FUNCTION "mb_internal_s" : Bool   // FC23, SCL
{ S7_Optimized_Access := 'TRUE' }
VERSION : 0.1
   VAR_INPUT
      start : DInt;
      end : DInt;
   END_VAR
   VAR_IN_OUT
      buffer_lo : DInt;
      buffer_hi : DInt;
      q : "mb_query";
   END_VAR
   VAR_TEMP
      tmp : DInt;
   END_VAR
BEGIN
   // Internal function in the library for calculating
   // beginning and end for swapping.
   // 
   // This function dosen't work for discrete quries !

   // Find the beginning in the buffer where swaping should start.
   #buffer_lo := SEL(G := #start = 0,
                     IN0 := (#start - UDINT_TO_DINT(#q.z.q.data_addr)) * 2,
                     IN1 := 0);

   // Find end point in buffer.
   IF #end = 0 THEN  // Auto - Swap all words in query.
       #buffer_hi := #q.z.q.data_len * 2 - 1;

   ELSE // Address given for #end.
       #buffer_hi := (#end - UDINT_TO_DINT(#q.z.q.data_addr)) * 2 - 1 ;
   END_IF;

   // Test if there is valid input values.
   #mb_internal_s := #buffer_lo >= 0 AND #buffer_hi <= 249 ;

   // Error handling.
   IF NOT #mb_internal_s THEN // If not valid values.
       #q.stat.status := 16#fffe;
       #q.Error := #q.stat.error := true;
       #q.Done := #q.stat.done := false;
       #q.z.sb.log_data_addr := #q.z.q.data_addr;
   END_IF;
END_FUNCTION

// folder: Library/Modbus/Core/z/z internal testing functions/z Testing

FUNCTION_BLOCK "tcp_test"   // FB96, SCL
{ S7_Optimized_Access := 'TRUE' }
VERSION : 0.1
   VAR
      mb_query : "mb_query";
      mb_client_ctrl : "mb_client_ctrl";
      t1 : Word;
      t2 : Word;
      t3 : Word;
      t4 : Word;
      aa : Bool;
      mb_delay_between_queries : "mb_delay_between_queries";
      sb : "mb_station_block_udt";
   END_VAR
BEGIN

   #mb_client_ctrl.ip_addr[1] := 192;
   #mb_client_ctrl.ip_addr[2] := 168;
   #mb_client_ctrl.ip_addr[3] := 0;
   #mb_client_ctrl.ip_addr[4] := 33;
   #mb_client_ctrl(interface := 64,
                   conn_id := 123,
                   tcp_port := 502,
                   // timeout := T#500ms,
                   mb_query := #mb_query);

   #mb_delay_between_queries(// delay := T#1s,
                             mb_query := #mb_query);

   "mb_station_block_header"(sb := #sb, mb_query := #mb_query);

   #mb_query(mb_addr := 255,
             mode := #mb_query.c.write.holding_reg,
             data_addr := 1,
             data_ptr := #t1);

   #mb_query(mode := #mb_query.c.read.holding_reg,
             data_addr := 1,
             data_ptr := #t2);

   #mb_query(mode := #mb_query.c.write.holding_reg,
             data_addr := 2,
             data_ptr := #t2);

   #mb_query(mode := #mb_query.c.read.holding_reg,
             data_addr := 2,
             data_ptr := #t3);

   "mb_station_block_footer"(sb := #sb, mb_query := #mb_query);
END_FUNCTION_BLOCK

FUNCTION_BLOCK "rtu_test_1500"   // FB102, SCL
{ S7_Optimized_Access := 'TRUE' }
VERSION : 0.1
   VAR
      mb_master_1500_ctrl : "mb_master_1500_ctrl";
      mb_query : "mb_query";
      temperature_1 : "Jdrk_RS_WS_N01_8";
      temperature_2 : "Jdrk_RS_WS_N01_8";
      temperature_3 : "Jdrk_RS_WS_N01_8";
      sb_temp_no_answer_1 : "sb_temp_no_answer";
      sb_temp_no_answer_2 : "sb_temp_no_answer";
      sb_temp_no_answer_3 : "sb_temp_no_answer";
      sb_temp_error_1 : "sb_temp_error";
      sb_temp_error_2 : "sb_temp_error";
      sb_temp_error_3 : "sb_temp_error";
      delay_between_queries : "mb_delay_between_queries";
      mb_delay : "mb_delay";
   END_VAR
BEGIN

   #mb_master_1500_ctrl.conf.parity := 0;
   #mb_master_1500_ctrl(hardware_id := 269,
                        operating_mode := 4,
                        baud := 9600,
                        mb_query := #mb_query);

   #delay_between_queries(mb_query := #mb_query);


   #temperature_1(mb_query := #mb_query);
   #temperature_2(mb_query := #mb_query);
   #temperature_3(mb_query := #mb_query);

   #mb_delay(mb_query := #mb_query);

   #sb_temp_no_answer_1(mb_query := #mb_query);
   #sb_temp_no_answer_2(mb_query := #mb_query);
   #sb_temp_no_answer_3(mb_query := #mb_query);

   #sb_temp_error_1(mb_query := #mb_query);
   #sb_temp_error_2(mb_query := #mb_query);
   #sb_temp_error_3(mb_query := #mb_query);
END_FUNCTION_BLOCK

FUNCTION_BLOCK "rtu_test2_1200"   // FB115, SCL
{ S7_Optimized_Access := 'TRUE' }
VERSION : 0.1
   VAR
      mb_query : "mb_query";
      mb_master_1200_ctrl : "mb_master_1200_ctrl";
      Danfoss : "Danfoss_VLT";
      Mjk_expert_1 : "Mjk_expert";
      Mjk_expert_2 : "Mjk_expert";
      Mjk_expert_3 : "Mjk_expert";
   END_VAR
BEGIN
   #mb_master_1200_ctrl.conf.parity := 0;
   #mb_master_1200_ctrl(hardware_id := 0, // "Local~CB_1241_(RS485)",
                        baud := 9600,
                        mb_query := #mb_query);

   #Mjk_expert_1(mb_addr := 1, mb_query := #mb_query);
   #Mjk_expert_2(mb_addr := 1, mb_query := #mb_query);
   #Mjk_expert_3(mb_addr := 1, mb_query := #mb_query);

   #Danfoss(mb_addr := 2, mb_query := #mb_query);
END_FUNCTION_BLOCK

FUNCTION_BLOCK "rtu_test1_1200"   // FB116, SCL
{ S7_Optimized_Access := 'TRUE' }
VERSION : 0.1
   VAR
      mb_query : "mb_query";
      mb_master_1200_ctrl : "mb_master_1200_ctrl";
      delay_between_queries : "mb_delay_between_queries";
      delay : "mb_delay";
      __ : Bool;
      temperature_1 : "Jdrk_RS_WS_N01_8";
      temperature_2 : "Jdrk_RS_WS_N01_8";
      temperature_3 : "Jdrk_RS_WS_N01_8";
      sb_temp_no_answer_1 : "sb_temp_no_answer";
      sb_temp_no_answer_2 : "sb_temp_no_answer";
      sb_temp_no_answer_3 : "sb_temp_no_answer";
      sb_temp_error_1 : "sb_temp_error";
      sb_temp_error_2 : "sb_temp_error";
      sb_temp_error_3 : "sb_temp_error";
      _ : Bool;
      bool_arrary : Array[0..15] of Bool;
      sb : "mb_station_block_udt";
   END_VAR
BEGIN
   #mb_master_1200_ctrl.conf.parity := 0;
   #mb_master_1200_ctrl(hardware_id := 269, // "Local~CB_1241_(RS485)",
                        baud := 9600,
                        mb_query := #mb_query);

   #delay_between_queries(mb_query := #mb_query);

   #temperature_1(mb_query := #mb_query);
   #temperature_2(mb_query := #mb_query);
   #temperature_3(mb_query := #mb_query);

   #delay(mb_query := #mb_query);

   #sb_temp_no_answer_1(mb_query := #mb_query);
   #sb_temp_no_answer_2(mb_query := #mb_query);
   #sb_temp_no_answer_3(mb_query := #mb_query);

   #sb_temp_error_1(mb_query := #mb_query);
   #sb_temp_error_2(mb_query := #mb_query);
   #sb_temp_error_3(mb_query := #mb_query);

   "mb_station_block_header"(sb := #sb, mb_query := #mb_query);
   #mb_query.mb_addr := 1;
   #mb_query.mode := #mb_query.c.read.input_reg;
   #mb_query.data_addr := 1;
   "mb_query_bits"(data_ptr := #bool_arrary, mb_query := #mb_query);
   "mb_station_block_footer"(sb := #sb, mb_query := #mb_query);
END_FUNCTION_BLOCK

// folder: Library/Modbus/Core/z/z internal testing functions/z Testing/nolib

FUNCTION_BLOCK "client"   // FB112, SCL
{ S7_Optimized_Access := 'TRUE' }
VERSION : 0.1
   VAR
      client : MB_CLIENT;
      tcon_ip_v4 : TCON_IP_v4;
      buffer : Array[0..3] of Byte;
      rtrig_err : R_TRIG;
      rtrig_busy : R_TRIG;
      rtrig_done : R_TRIG;
      err_cnt : UDInt;
      busy_cnt : UDInt;
      done_cnt : UDInt;
      a4 : USInt;
   END_VAR
BEGIN
   #tcon_ip_v4.InterfaceId := 64;
   #tcon_ip_v4.ID := 456;
   #tcon_ip_v4.ConnectionType := 11; // tcp
   #tcon_ip_v4.ActiveEstablished := true;
   #tcon_ip_v4.RemoteAddress.ADDR[1] := 192;
   #tcon_ip_v4.RemoteAddress.ADDR[2] := 168;
   #tcon_ip_v4.RemoteAddress.ADDR[3] := 0;
   #tcon_ip_v4.RemoteAddress.ADDR[4] := #a4;
   #tcon_ip_v4.RemotePort := 502;

   #client(REQ := #client.REQ,
           DISCONNECT := #client.DISCONNECT,
           MB_MODE := 103,
           MB_DATA_ADDR := 1000,
           MB_DATA_LEN := 1,
           MB_DATA_PTR := #buffer,
           CONNECT := #tcon_ip_v4);

   #rtrig_err(CLK := #client.ERROR);
   #err_cnt += BOOL_TO_UINT( #rtrig_err.Q );

   #rtrig_busy(CLK := #client.BUSY);
   #busy_cnt += BOOL_TO_UINT(#rtrig_busy.Q);

   #rtrig_done(CLK := #client.DONE);
   #done_cnt += BOOL_TO_UINT(#rtrig_done.Q);
END_FUNCTION_BLOCK

// folder: Library/Modbus/Core/z/z internal testing functions/z Testing/sb

FUNCTION_BLOCK "sb_temp_no_answer"   // FB32, SCL
{ S7_Optimized_Access := 'TRUE' }
VERSION : 0.1
   VAR_OUTPUT
      Temperature : Real;
   END_VAR
   VAR_IN_OUT
      mb_query : "mb_query";
   END_VAR
   VAR
      sb : "mb_station_block_udt";
   END_VAR
   VAR RETAIN
      offset : Real;
   END_VAR
   VAR_TEMP
      tmp : Int;
   END_VAR
BEGIN
   // JDRK - RS-WS-N01-8 - Temperature and Humidity sensor

   "mb_station_block_header"(sb := #sb, mb_query := #mb_query);

   #mb_query(mb_addr := 200,
             mode := #mb_query.c.read.input_reg,
             data_addr := 1,
             data_ptr := #tmp);

   IF #mb_query.Done THEN
       #Temperature := INT_TO_REAL(#tmp) / 10 + #offset;
   END_IF;

   "mb_station_block_footer"(sb := #sb, mb_query := #mb_query);
END_FUNCTION_BLOCK

FUNCTION_BLOCK "sb_temp_error"   // FB33, SCL
{ S7_Optimized_Access := 'TRUE' }
VERSION : 0.1
   VAR_OUTPUT
      Temperature : Real;
   END_VAR
   VAR_IN_OUT
      mb_query : "mb_query";
   END_VAR
   VAR
      sb : "mb_station_block_udt";
   END_VAR
   VAR RETAIN
      tt : Array[0..100] of Int;
   END_VAR
   VAR_TEMP
      tmp : Int;
   END_VAR
BEGIN
   // JDRK - RS-WS-N01-8 - Temperature and Humidity sensor

   "mb_station_block_header"(sb := #sb, mb_query := #mb_query);

   #mb_query(mb_addr := 1,
             mode := #mb_query.c.read.input_reg,
             data_addr := 1,
             data_ptr := #tmp);

   IF #mb_query.Done THEN
       #Temperature := INT_TO_REAL(#tmp) / 10;
   END_IF;

   // Query producing a error.
   #mb_query(mb_addr := 1,
             mode := #mb_query.c.read.input_reg,
             data_addr := 1,
             data_ptr := #tt);

   "mb_station_block_footer"(sb := #sb, mb_query := #mb_query);
END_FUNCTION_BLOCK

// folder: Library/Modbus/Core/z Special code snippets examples/Not needed for regular users

FUNCTION_BLOCK "Example Done and error"   // FB56, SCL
{ S7_Optimized_Access := 'TRUE' }
VERSION : 0.1
   VAR_IN_OUT
      mb_query : "mb_query";
   END_VAR
   VAR
      query1_data : Word;
      done_cnt : UInt;
      query2_data : Word;
   END_VAR
BEGIN
   // To get information about when a particular query has executed.

   #mb_query(mb_addr := 123,
             mode := #mb_query.c.write.holding_reg,
             data_addr := 456,
             data_ptr := #query1_data);

   // The if-statement bellow has to be put after the particular 
   // query, and before the next query.    

   IF #mb_query.Done THEN
       // Some action after a successfully query.    
       #done_cnt += 1; // Eg. count successfully queries.

   ELSIF #mb_query.Error THEN
       // Some action if a faild query.    

       // #mb_query.stat.status , gives more information about 
       // the error.         

       IF #mb_query.stat.error_comm THEN
           ; // Some particular action if communication error.
       END_IF;

   END_IF;

   // Next query...
   #mb_query(mb_addr := 111,
             mode := #mb_query.c.read.holding_reg,
             data_addr := 789,
             data_ptr := #query2_data);
END_FUNCTION_BLOCK

FUNCTION_BLOCK "Example Swap"   // FB78, SCL
{ S7_Optimized_Access := 'TRUE' }
VERSION : 0.1
   VAR_IN_OUT
      mb_query : "mb_query";
   END_VAR
   VAR
      static_tmp_var : DWord;
      value : DWord;
      value2 : DWord;
      value_real_1 : Real;
      value_real_2 : Real;
   END_VAR
   VAR_TEMP
      "e" : Int;
      param : "mb_set_udt";
   END_VAR
   VAR CONSTANT
      ALL : Int;
   END_VAR
BEGIN
   // For some modbus devices, when two registers are combined into one,
   // the data is stored as little endian, not big endian like Siemens 
   // PLC does. To solve this, the SWAP function needs to be utilized.
   #mb_query(mb_addr := 123,
             mode := #mb_query.c.read.holding_reg,
             data_addr := 123,
             data_ptr := #static_tmp_var);

   #value := SWAP(#static_tmp_var);


   // For other device, when two registers are combined, the least significant 
   // word is stored first and the most significant word is stored in the 
   // following register. When this is the case, the ROR-function needs 
   // to be used.
   #mb_query(mb_addr := 123,
             mode := #mb_query.c.read.holding_reg,
             data_addr := 123,
             data_ptr := #static_tmp_var);

   #value := ROR(IN := #static_tmp_var, N := 16);


   // In some situation both SWAP and ROR need to be used.
   #mb_query(mb_addr := 123,
             mode := #mb_query.c.read.holding_reg,
             data_addr := 123,
             data_ptr := #static_tmp_var);

   #value := SWAP(ROR(IN := #static_tmp_var, N := 16));

   // How the data is stored, is usually described in the
   // data sheet of each device.

   // ========================================================================

   // The code bellow it's anather approach. It may be har understand, but it 
   // should be okay to understand what it do.

   IF "mb_query_range"(start := 100, end := 150, q := #mb_query) THEN
       #"e" := "mb_swap_word"(start := #ALL, end := #ALL, q := #mb_query);
       #"e" := "mb_read_buffer"(addr := 100, ptr := #value, q := #mb_query);
       #"e" := "mb_read_buffer"(addr := 120, ptr := #value2, q := #mb_query);
   END_IF;

   IF "mb_query_range"(start := 200, end := 250, q := #mb_query) THEN
       #param.double := true; // 4 bytes
       #param.factor := 10; // 
       #value_real_1 := "mb_buffer_get"(addr := 200, param := #param, q := #mb_query);
       #value_real_2 := "mb_buffer_get"(addr := 220, param := #param, q := #mb_query);
   END_IF;
END_FUNCTION_BLOCK

FUNCTION_BLOCK "Example Read first"   // FB85, SCL
{ S7_Optimized_Access := 'TRUE' }
VERSION : 0.1
   VAR_INPUT
      input1 : Bool;
      input2 : Bool;
   END_VAR
   VAR_IN_OUT
      mb_query : "mb_query";
   END_VAR
   VAR
      write : Bool;
      data : Word;
   END_VAR
BEGIN
   // Sometimes only some bits in a word need to be manipulated, 
   // without touching the other bits, bellow is an example how 
   // that can be achieved.

   #mb_query.mb_addr := 123;
   #mb_query.data_addr := 456;

   IF #write THEN // (Initially false)

       // Manipulating only bit 5 and 11
       #data.%X5 := #input1;
       #data.%X11 := #input2;

       #mb_query(mode := #mb_query.c.write.holding_reg,
                 data_ptr := #data);

   ELSE // read the register before write to the same one.
       #mb_query(mode := #mb_query.c.read.holding_reg,
                 data_ptr := #data);

       // Has query above been executed successfully?
       IF #mb_query.Done THEN
           #write := true;
       END_IF;

   END_IF;

   // Note: The read only option (#sb.conf.read_conly) can't be
   // used when the metod above is used.
END_FUNCTION_BLOCK

FUNCTION_BLOCK "Example Forced execution order"   // FB89, SCL
{ S7_Optimized_Access := 'TRUE' }
VERSION : 0.1
   VAR_IN_OUT
      mb_query : "mb_query";
   END_VAR
   VAR
      state : Int;
      query_1 : Word;
      query_2 : UInt;
      query_3 : Word;
      query_4 : Word;
   END_VAR
BEGIN
   // If the execution need to be forced to a given order, then the 
   // example bellow can be followed.

   CASE #state OF

       0:  // 1st query
           #mb_query(mb_addr := 123,
                     mode := #mb_query.c.write.holding_reg,
                     data_addr := 123,
                     data_ptr := #query_1);
           #state += BOOL_TO_SINT(#mb_query.Done);
           // «#mb_query.done» is set true when the query above is done 
           // successfully. When next query is executed, «#mb_query.done»
           // is set back false.

       1:  // 2nd query
           #mb_query(mb_addr := 123,
                     mode := #mb_query.c.write.holding_reg,
                     data_addr := 456,
                     data_ptr := #query_2);
           #state += BOOL_TO_SINT(#mb_query.Done);

       2:  // 3rd query
           #mb_query(mb_addr := 123,
                     mode := #mb_query.c.read.holding_reg,
                     data_addr := 789,
                     data_ptr := #query_3);
           IF #mb_query.Done THEN
               #state := 0;
           END_IF;

   END_CASE;

   // 4th query, this query is executed three times as often 
   // as the queries above.
   #mb_query(mb_addr := 123,
             mode := #mb_query.c.read.input_reg,
             data_addr := 1234,
             data_ptr := #query_4);


   // If the state machine has both read and write queries then
   // #sb.conf.read_only can't be used.
END_FUNCTION_BLOCK

FUNCTION_BLOCK "Example discrete queries"   // FB101, SCL
{ S7_Optimized_Access := 'TRUE' }
VERSION : 0.1
   VAR_IN_OUT
      mb_query : "mb_query";
   END_VAR
   VAR
      one_bool : Bool;
      two_bools : Struct
         b1 : Bool;
         b2 : Bool;
      END_STRUCT;
   END_VAR
BEGIN
   // Discrete queries.

   // When doing discrete queries the data_len parameter need to
   // be specified manualy.
   #mb_query(mb_addr := 123,
             mode := #mb_query.c.read.discrete_input,
             data_addr := 456,
             data_len := 1,
             data_ptr := #one_bool); // A single boolean.

   // Another quering two bool's
   #mb_query(mb_addr := 123,
             mode := #mb_query.c.read.discrete_input,
             data_addr := 789,
             data_len := 2,
             data_ptr := #two_bools); // A struct with two boolean inside.

   // After discrete queries, data_len should be set back in to auto.
   #mb_query.data_len := #mb_query.c.auto_len;
END_FUNCTION_BLOCK

FUNCTION_BLOCK "Example sequence"   // FB103, SCL
{ S7_Optimized_Access := 'TRUE' }
VERSION : 0.1
   VAR_INPUT
      mb_addr : USInt;
   END_VAR
   VAR_IN_OUT
      mb_query : "mb_query";
   END_VAR
   VAR
      sb : "mb_station_block_udt";
      sequence : "mb_sequence";
      read1 : Word;
      read2 : Word;
      read3 : Word;
      write1 : Word;
      write2 : Word;
      write3 : Word;
   END_VAR
BEGIN
   "mb_station_block_header"(sb := #sb, mb_query := #mb_query);
   #mb_query.mb_addr := #mb_addr;

   // High priority queries:
   #mb_query(mode := #mb_query.c.read.holding_reg,
             data_addr := 12345,
             data_ptr := #write3);

   IF #sequence.Done THEN
       #mb_query(mode := #mb_query.c.write.holding_reg,
                 data_addr := 54321,
                 data_ptr := #write3);
   END_IF;

   // Low priority queries:
   // Some queries that doesn't need to be run so often, the state
   // machines bellow make low priority queries be executed less often.
   #sequence.conf.first_state := 1600;
   CASE "mb_sequence_init"(sequence := #sequence, mb_query := #mb_query) OF
           // --------- Read holding reg queries (3xx) ---------
       300: #mb_query(data_addr := 123, data_ptr := #read1);
       301: #mb_query(data_addr := 456, data_ptr := #read2);
       302: #mb_query(data_addr := 789, data_ptr := #read3);

           #sequence.next_state := 1600;
           // --------- Write holding reg queries (16xx) ---------     
       1600: #mb_query(data_addr := 654, data_ptr := #write1);
       1601: #mb_query(data_addr := 321, data_ptr := #write2);
           #sequence.next_state := 300;
       ELSE
           #sequence.state += 1;
   END_CASE;
   #sequence(sb := #sb, mb_query := #mb_query);

   "mb_station_block_footer"(sb := #sb, mb_query := #mb_query);
END_FUNCTION_BLOCK

// folder: Library/Modbus/Docs

FUNCTION "mb_version" : String   // FC6, SCL
{ S7_Optimized_Access := 'TRUE' }
VERSION : 0.1
BEGIN
   // Library version.
   #mb_version := '3.2.0';

   (*

   www.rexhip.com


   Copyright (c) 2018 Ola Bjørnli 

   Permission is hereby granted, free of charge, to any person obtaining a copy
   of this software and associated documentation files (the "Software"), to deal
   in the Software without restriction, including without limitation the rights
   to use, copy, modify, merge, publish, distribute, sublicense, and/or sell
   copies of the Software, and to permit persons to whom the Software is
   furnished to do so, subject to the following conditions:

   The above copyright notice and this permission notice shall be included in all
   copies or substantial portions of the Software.

   THE SOFTWARE IS PROVIDED "AS IS", WITHOUT WARRANTY OF ANY KIND, EXPRESS OR
   IMPLIED, INCLUDING BUT NOT LIMITED TO THE WARRANTIES OF MERCHANTABILITY,
   FITNESS FOR A PARTICULAR PURPOSE AND NONINFRINGEMENT. IN NO EVENT SHALL THE
   AUTHORS OR COPYRIGHT HOLDERS BE LIABLE FOR ANY CLAIM, DAMAGES OR OTHER
   LIABILITY, WHETHER IN AN ACTION OF CONTRACT, TORT OR OTHERWISE, ARISING FROM,
   OUT OF OR IN CONNECTION WITH THE SOFTWARE OR THE USE OR OTHER DEALINGS IN THE
   SOFTWARE.

   *)
END_FUNCTION

FUNCTION "mb_Debugging" : Void   // FC15, SCL
{ S7_Optimized_Access := 'TRUE' }
VERSION : 0.1
BEGIN
   (* 
   # General debugging:
   - Look online and check that the latest version of the library 
     is in use. (www.rexhip.com or github.com/rexhip/rexhip)
   - All queries need to be executed in same order, this implicates 
     that it's NOT possible to put some queries in interupts and 
     other in cyclic OB's, this would interfere with the order.
   - Look inside the data blcok of the SB of the device that having 
     problem, and locate «#sb.log...», see if the counters are 
     running and lookup the error code of «#sb.log.error_status», 
     «#sb.log.error_data_addr» will tell witch query generating the 
     error. 
   - Try reboot PLC.

   # Modbus RTU
   - Try to increase timeout, repeaters on the bus need additional 
     time.
   - All the devies on the bus need to have a unique address.
   - Parity, buard rate, stop bits need to be the same in all 
     devices. The modbus specification state on page 20, that 19200
     is the default/recommended buad rate. The specification also 
     state, on page 12, that parity should be "even".
   - Electrical polarity, for some devices the connection "A" and "B" 
     is mislabeled, try to swap them.
   - Check for correct hardware id,

   # Modbus TCP
   - Try to increase timeout, creating a TCP-connection may take long.
   - Check IP-address.
   - Check TCP-port, 502 is default.
   - Check for unic connection-id.
   - Try set unit address to 255, (not for gateways)

   # Station Blocks 
   - If mb_station_block_header has executed in one block then 
     mb_station_block_foother also need to be executed. Cheack that 
     there is no RETURN or simular between them.
   - Check datasheet of device for special requirement: function codes 
     supported, max data length, register required to be queried 
     together, etc.  
   - A query can't be longer then 124 words.   
   - Try to comment out queries and see if it solve the problem.  

   # TIA-portal upgrading firmware error
     If you upgrade the firmware of a plc in a project, several errors in 
     the code regarding in serialize and deserialize will appear. This is 
     due to a error in TIA-portal. The solution is avoid using the upgrade 
     function, and rather add a new plc in the project and move all 
     elements to the new plc.

   # Some status codes and solutions:
     8188:     Try upgrade to latest version of the library. 

   # Customs status error codes
   - ffff: mb_read_buffer:     The request data is not avalible inside the 
                               buffer. check value of #addr.                            
   - fffe:                     
   - fffd: mb_buffer_get       The request data is not avalible inside the 
                               buffer. check value of #addr.

   *)
END_FUNCTION

// folder: Library/Modbus/Station blocks/sb Tested/Danfoss

FUNCTION_BLOCK "Danfoss_VLT"   // FB71, SCL
{ S7_Optimized_Access := 'TRUE' }
VERSION : 0.1
   VAR_INPUT
      mb_addr : USInt;
   END_VAR
   VAR_IN_OUT
      mb_query : "mb_query";
   END_VAR
   VAR
      sb : "mb_station_block_udt";
   END_VAR
   VAR RETAIN
      conf : Struct
         Send_config_to_drive : Bool := true;
         auto_start : Bool;
         action_no_communication : Int := 2;   // 2: Stop,
         input_source : Int := 2;   // 2: ctw fieldbus
      END_STRUCT;
   END_VAR
   VAR
      data : "variable_frequency_drive_udt";
      alarm_word : DWord;
      read : Struct   // (unscaled)
         stw : Struct   // Status word
            speed_eq_reference : Bool;   // [08]
            bus_control : Bool;   // [09] false=hand mode
            frequency_limit_ok : Bool;   // [10]
            in_operation : Bool;   // [11]
            stopped_auto_start : Bool;   // [12]
            voltage_exceeded : Bool;   // [13]
            torque_exceeded : Bool;   // [14]
            timer_exceeded : Bool;   // [15]
            control_ready : Bool;   // [00]
            drive_ready : Bool;   // [01]
            enable : Bool;   // [02] 0=Coasting
            trip : Bool;   // [03]
            error_no_trip : Bool;   // [04]
            x05 : Bool;   // [05]
            triplock : Bool;   // [06]
            warning : Bool;   // [07]
         END_STRUCT;
         man : Int;   // man actual value
      END_STRUCT;
      write : Struct   // Controll word
         ctw : Struct   // Controll word
            x08 : Bool;   // [08]
            use_ramp_2 : Bool;   // [09]
            data_valid : Bool := TRUE;   // [10]
            x11 : Bool;   // [11]
            x12 : Bool;   // [12]
            x13 : Bool;   // [13]
            x14 : Bool;   // [14]
            reverse : Bool;   // [15]
            x00 : Bool;   // [00]
            x01 : Bool;   // [01]
            dc_break_NOT : Bool := TRUE;   // [02]
            coast_NOT : Bool := TRUE;   // [03]
            quick_stop_NOT : Bool := TRUE;   // [04]
            hold_output_frequency_NOT : Bool := TRUE;   // [05]
            start : Bool;   // [06]
            reset : Bool;   // [07]
         END_STRUCT;
         ref : Int;
      END_STRUCT;
      sequence : "mb_sequence";
   END_VAR
   VAR_TEMP
      tmp : Int;
      dtmp : DInt;
   END_VAR
BEGIN
   (*  Danfoss - VLT
       doc_MG20N202.pdf, doc_MG20O602.pdf

       8.4 : Action if no communication.    (2=stop)     
       8.1 : Select input source            (2=CTW=fieldbus)     
   *)
   "mb_station_block_header"(sb := #sb, mb_query := #mb_query);
   #mb_query.mb_addr := #mb_addr;

   REGION Low priority queries
       // Some queries that doesn't need to be run so often, the state machines
       // bellow make low priority queries be executed less often.
       #sequence.conf.first_state := SEL(G := #conf.Send_config_to_drive,
                                         IN0 := 300, IN1 := 1600);
       CASE "mb_sequence_init"(sequence := #sequence, mb_query := #mb_query) OF
               // --------- Read holding reg queries ---------
           300:  // Frequency (hz)
               #mb_query(data_addr := "p"(a := 16, b := 13), data_ptr := #tmp);
               IF #mb_query.Done THEN
                   #data.out.frequency := DINT_TO_REAL(#tmp) * 0.1;
               END_IF;
           301:  // Electrical current 
               #mb_query(data_addr := "p"(a := 16, b := 14), data_ptr := #dtmp);
               IF #mb_query.Done THEN
                   #data.out.current := DINT_TO_REAL(#dtmp) * 0.01;
               END_IF;
           302:  // RPM
               #mb_query(data_addr := "p"(a := 16, b := 17), data_ptr := #dtmp);
               IF #mb_query.Done THEN
                   #data.out.rpm := DINT_TO_REAL(#dtmp) / 60;
               END_IF;
           303:  // Power
               #mb_query(data_addr := "p"(a := 16, b := 10), data_ptr := #dtmp);
               IF #mb_query.Done THEN
                   #data.out.power := DINT_TO_REAL(#dtmp) * 10;
               END_IF;
           304:  // Heatsink Temp. 
               #mb_query(data_addr := "p"(a := 16, b := 34), data_ptr := #tmp);
               IF #mb_query.Done THEN
                   #data.out.heatsing_temperature := #tmp;
               END_IF;
           305:  // Motor voltage
               #mb_query(data_addr := "p"(a := 16, b := 12), data_ptr := #tmp);
               IF #mb_query.Done THEN
                   #data.out.voltage := INT_TO_REAL(#tmp) * 0.1;
               END_IF;
           306:  // Alarm word 
               #mb_query(data_addr := "p"(a := 16, b := 92), data_ptr := #dtmp);
               IF #mb_query.Done THEN
                   #alarm_word := DINT_TO_DWORD(#dtmp);
               END_IF;
           307:  // Torque [%] 
               #mb_query(data_addr := "p"(a := 16, b := 22), data_ptr := #tmp);
               IF #mb_query.Done THEN
                   #data.out.torque_percent := #tmp;
               END_IF;
               #sequence.next_state := #sequence.conf.first_state;

               // --------- Write holding reg queries ---------     
           1600: // Action if no communication. (2=stop)     
               #mb_query(data_addr := "p"(a := 8, b := 4),
                         data_ptr := #conf.action_no_communication);
           1601: // Select input source (2=CTW=fieldbus)     
               #mb_query(data_addr := "p"(a := 8, b := 1),
                         data_ptr := #conf.input_source);
               #sequence.next_state := 300;
           ELSE
               #sequence.state += 1;
       END_CASE;
       #sequence(sb := #sb, mb_query := #mb_query);
   END_REGION

   REGION High priority queries
       // Status word  and main actual value 
       #mb_query(mode := #mb_query.c.read.holding_reg,
                 data_addr := 2909,
                 data_ptr := #read);
       IF #mb_query.Done THEN
           #data.out.ready := #read.stw.control_ready
           (* *)AND #read.stw.drive_ready AND #read.stw.bus_control;
           #data.out.error := #read.stw.trip OR #read.stw.error_no_trip;
           #data.out.auto := #read.stw.bus_control;
           #data.out.in_operation := #read.stw.in_operation;
           #data.out.output_percent := INT_TO_REAL(#read.man) / 16#4000 * 100;
       END_IF;
       // Send ctw and ref
       #write.ctw.reset := #data.in.reset;
       #write.ctw.dc_break_NOT := NOT #data.in.dc_break;
       #write.ctw.coast_NOT := NOT #data.in.cost;
       #write.ctw.quick_stop_NOT := NOT #data.in.quick_stop;
       #write.ctw.start := #data.in.start;
       #write.ref := REAL_TO_INT(#data.in.ref / 100 * 16#4000);
       #mb_query(mode := #mb_query.c.write.holding_reg,
                 data_addr := 2809,
                 data_ptr := #write);
   END_REGION

   "mb_station_block_footer"(sb := #sb, mb_query := #mb_query);

   (* Terminals:
   68  RS485 D+
   69  RS485 D-
   *)
END_FUNCTION_BLOCK

FUNCTION_BLOCK "Danfoss_VLT_simple"   // FB124, SCL
{ S7_Optimized_Access := 'TRUE' }
VERSION : 0.1
   VAR_INPUT
      mb_addr : USInt;
      ref : Real;
      start : Bool;
      cost : Bool;
      dc_break : Bool;
      quick_stop : Bool;
   END_VAR
   VAR_OUTPUT
      Ready : Bool;
      Feedback : Real;
   END_VAR
   VAR_IN_OUT
      mb_query : "mb_query";
   END_VAR
   VAR
      sb : "mb_station_block_udt";
      data : "variable_frequency_drive_udt";
      read : Struct   // (unscaled)
         stw : Struct   // Status word
            speed_eq_reference : Bool;   // [08]
            bus_control : Bool;   // [09] false=hand mode
            frequency_limit_ok : Bool;   // [10]
            in_operation : Bool;   // [11]
            stopped_auto_start : Bool;   // [12]
            voltage_exceeded : Bool;   // [13]
            torque_exceeded : Bool;   // [14]
            timer_exceeded : Bool;   // [15]
            control_ready : Bool;   // [00]
            drive_ready : Bool;   // [01]
            enable : Bool;   // [02] 0=Coasting
            trip : Bool;   // [03]
            error_no_trip : Bool;   // [04]
            x05 : Bool;   // [05]
            triplock : Bool;   // [06]
            warning : Bool;   // [07]
         END_STRUCT;
         man : Int;   // man actual value
      END_STRUCT;
      write : Struct   // Controll word
         ctw : Struct   // Controll word
            x08 : Bool;   // [08]
            use_ramp_2 : Bool;   // [09]
            data_valid : Bool := TRUE;   // [10]
            x11 : Bool;   // [11]
            x12 : Bool;   // [12]
            x13 : Bool;   // [13]
            x14 : Bool;   // [14]
            reverse : Bool;   // [15]
            x00 : Bool;   // [00]
            x01 : Bool;   // [01]
            dc_break_NOT : Bool := TRUE;   // [02]
            coast_NOT : Bool := TRUE;   // [03]
            quick_stop_NOT : Bool := TRUE;   // [04]
            hold_output_frequency_NOT : Bool := TRUE;   // [05]
            start : Bool;   // [06]
            reset : Bool;   // [07]
         END_STRUCT;
         ref : Int;
      END_STRUCT;
   END_VAR
BEGIN
   (*  Danfoss - VLT
       doc_MG20N202.pdf, doc_MG20O602.pdf

       8.4 : Action if no communication.    (2=stop)     
       8.1 : Select input source            (2=CTW=fieldbus)     

       Terminals:
       68  RS485 D+
       69  RS485 D-
   *)
   "mb_station_block_header"(sb := #sb, mb_query := #mb_query);
   #mb_query.mb_addr := #mb_addr;

   // Status word  and main actual value 
   #mb_query(mode := #mb_query.c.read.holding_reg,
             data_addr := 2909,
             data_ptr := #read);
   IF #mb_query.Done THEN
       #Ready := #read.stw.control_ready
       (* *)AND #read.stw.drive_ready AND #read.stw.bus_control;
       #Feedback := INT_TO_REAL(#read.man) / 16#4000 * 100;
   END_IF;

   // Send ctw and ref
   #write.ctw.dc_break_NOT := NOT #dc_break;
   #write.ctw.coast_NOT := NOT #cost;
   #write.ctw.quick_stop_NOT := NOT #quick_stop;
   #write.ctw.start := #start;
   #write.ref := REAL_TO_INT(#ref / 100 * 16#4000);
   #mb_query(mode := #mb_query.c.write.holding_reg,
             data_addr := 2809,
             data_ptr := #write);

   "mb_station_block_footer"(sb := #sb, mb_query := #mb_query);
END_FUNCTION_BLOCK

FUNCTION "p" : UInt   // FC14, SCL
{ S7_Optimized_Access := 'TRUE' }
VERSION : 0.1
   VAR_INPUT
      "a" : USInt;
      "b" : USInt;
   END_VAR
BEGIN
   // Calculation data_addr for danfoss vlt.

   #p := USINT_TO_UINT(#"a") * 1000
   (* *)+ USINT_TO_UINT(#"b") * 10
   (* *)- 1;
END_FUNCTION

// folder: Library/Modbus/Station blocks/sb Tested/MJK

FUNCTION_BLOCK "Mjk_expert"   // FB35, SCL
{ S7_Optimized_Access := 'TRUE' }
VERSION : 0.1
   VAR_INPUT
      mb_addr : USInt;
   END_VAR
   VAR_IN_OUT
      mb_query : "mb_query";
   END_VAR
   VAR
      sb : "mb_station_block_udt";
      data : Struct
         pressure : Real;
         temperature : Real;
      END_STRUCT;
   END_VAR
BEGIN
   // MJK - Expert 700-7060-7070 - Pressure transmitters

   "mb_station_block_header"(sb := #sb, mb_query := #mb_query);
   #mb_query.mb_addr := #mb_addr;

   #mb_query.mode := #mb_query.c.read.holding_reg;
   #mb_query(data_addr := 16#100, data_ptr := #data);

   "mb_station_block_footer"(sb := #sb, mb_query := #mb_query);

   (*
       Rød     +24V
       Brown   GND
       Yellow  RS485 B
       Gray    RS485 A
       White   Voltage output
   *)
END_FUNCTION_BLOCK

// folder: Library/Modbus/Station blocks/sb Tested/Ponsel mesure

FUNCTION_BLOCK "Ponsel_mesure_Conductivity_C4E"   // FB105, SCL
{ S7_Optimized_Access := 'TRUE' }
VERSION : 0.1
   VAR_INPUT
      mb_addr : UInt := 255;   // 255=broadcast
   END_VAR
   VAR_OUTPUT
      Temperature : Real;   // [degree C]
      Conductivity : Real;   // [uS/cm]
      Salinity : Real;   // [ppt]
      TDS_Kcl : Real;   // [ppm]
      measurement_ok : Bool;
   END_VAR
   VAR_IN_OUT
      mb_query : "mb_query";
   END_VAR
   VAR
      ponsel_mesure : "Ponsel_mesure";
   END_VAR
   VAR_TEMP
      start : Bool;
   END_VAR
BEGIN
   // Ponsel mesure - Conductivity_C4E

   #start := true; // Continuous measurements

   #ponsel_mesure.minimum_measurement_interval := T#1s;
   #ponsel_mesure(mb_addr := #mb_addr,
                  compensate_enable := false,
                  Measurement_ok => #measurement_ok,
                  start_measurement := #start,
                  mb_query := #mb_query);

   #Temperature := #ponsel_mesure.data1.value[0];  // [degree C]
   #Conductivity := #ponsel_mesure.data1.value[1]; // [uS/cm]
   #Salinity := #ponsel_mesure.data1.value[2];     // [ppt]
   #TDS_Kcl := #ponsel_mesure.data1.value[3];      // [ppm]
END_FUNCTION_BLOCK

FUNCTION_BLOCK "Ponsel_mesure_Dissolved_oxygen"   // FB106, SCL
{ S7_Optimized_Access := 'TRUE' }
VERSION : 0.1
   VAR_INPUT
      mb_addr : UInt := 10;   // 255=broadcast
      start : Bool := TRUE;   // (Else use start to init messurements)
      measurement_interval : Time := T#1M;
      compensate_atmospheric_pressure : Real := 1013.0;   // hPa
      compensate_salinity : Real := 0.0;   // ppm
   END_VAR
   VAR_OUTPUT
      Temperature : Real;   // [degree C]
      Oxygen_Sat : Real;   // [%]
      Oxygen_mgl : Real;   // [mg/L]
      Oxygen_ppm : Real;   // [ppm]
      measurement_ok : Bool;
      serial_number : String[32];
   END_VAR
   VAR_IN_OUT
      mb_query : "mb_query";
   END_VAR
   VAR
      ponsel_mesure : "Ponsel_mesure";
   END_VAR
   VAR_TEMP
      start_measurement : Bool;
   END_VAR
BEGIN
   // Aqualabo - Ponsel mesure
   // Dissolved oxygen (OPTOD)
   // 
   // Warning: Each pull for sensor measurement, will reduce the available 
   // life span. Please set the measurement interval to appropriate value.

   #start_measurement := #start; // #measurement_interval will define intervals.

   #ponsel_mesure.minimum_measurement_interval := #measurement_interval;
   #ponsel_mesure.compensate[1] := #compensate_atmospheric_pressure;
   #ponsel_mesure.compensate[2] := #compensate_salinity;
   #ponsel_mesure(mb_addr := #mb_addr,
                  compensate_enable := true,
                  Measurement_ok => #measurement_ok,
                  start_measurement := #start_measurement,
                  mb_query := #mb_query);

   #Temperature := #ponsel_mesure.data1.value[0]; // [degree C]
   #Oxygen_Sat := #ponsel_mesure.data1.value[1];  // [%]
   #Oxygen_mgl := #ponsel_mesure.data1.value[2];  // [mg/l]
   #Oxygen_ppm := #ponsel_mesure.data1.value[3];  // [ppm]

   #serial_number := #ponsel_mesure.data2.serial_number;
END_FUNCTION_BLOCK

// folder: Library/Modbus/Station blocks/sb Tested/Ponsel mesure/Misc

FUNCTION_BLOCK "ponselMessure_ChangeMbAddr"   // FB94, SCL
{ S7_Optimized_Access := 'TRUE' }
VERSION : 0.1
   VAR_INPUT
      current_addr : USInt;
      new_addr : UInt;
      exec : Bool := TRUE;
   END_VAR
   VAR_OUTPUT
      Done : Bool;
      Error : Bool;
   END_VAR
   VAR_IN_OUT
      mb_query : "mb_query";
   END_VAR
   VAR_TEMP
      d : Bool;
      "e" : Bool;
   END_VAR
BEGIN
   IF #new_addr < 1 OR #new_addr > 247
       OR #new_addr = #current_addr
   THEN
       #"e" := TRUE;
   ELSIF #exec THEN
       #mb_query(mb_addr := #current_addr,
                 mode := #mb_query.c.write.holding_reg,
                 data_addr := 16#A3,
                 Done => #d,
                 Error => #"e",
                 data_ptr := #new_addr);
   END_IF;
   #Done := #d;
   #Error := #"e";
END_FUNCTION_BLOCK

FUNCTION_BLOCK "Ponsel_mesure"   // FB107, SCL
{ S7_Optimized_Access := 'TRUE' }
VERSION : 0.1
   VAR_INPUT
      mb_addr : UInt;
      minimum_measurement_interval : Time := T#1M;
      compensate_enable : Bool;
      compensate : Array[1..2] of Real;
   END_VAR
   VAR_OUTPUT
      Measurement_ok : Bool;
   END_VAR
   VAR_IN_OUT
      mb_query : "mb_query";
      start_measurement : Bool;
   END_VAR
   VAR
      sb : "mb_station_block_udt";
      QueryCnt : UDInt;
      data1 : Struct
         value : Array[0..4] of Real;
         compensate_temperature : Real;
         compensate : Array[1..2] of Real;
         _ : Word;
         status : Array[0..4] of Struct
            x08_StmGamme0 : Bool;
            x09_StmGamme1 : Bool;
            x10_StmGamme2 : Bool;
            x11 : Bool;
            x12 : Bool;
            x13 : Bool;
            x14 : Bool;
            x15 : Bool;
            x00_Stm0 : Bool;
            x01_Stm1 : Bool;
            x02_Stm2 : Bool;
            x03_StmTemp : Bool;   // At least one parameter coefficient uses a temporary calibration standard (configuration during calibration)
            x04_StmHF : Bool;   // At least one parameter coefficient is outside calibration limits
            x05_StmCU : Bool;   // All parameter coefficients use default coefficient
            x06_StmHIST : Bool;   // All parameter coefficients use history coefficient
            x07_StmME : Bool;   // Dry weight is missing in at least one parameter coefficient (measurement under way)
         END_STRUCT;
         Compensates_3 : Real;
      END_STRUCT;
      data2 : Struct
         Description : String[30];
         serial_number : String[32];   // (addr 0x0D10)
         Software_version : Word;   // Heavy Weight: Major version and Light Weight: Minor Version.
         Hardware_version : Word;   // Heavy Weight: Major version and Light Weight: Minor Version.
      END_STRUCT;
      api : Struct
         idle : Bool;
         wait : Bool;
         interval : Time;
      END_STRUCT;
      _ : Bool;   // Internal variables bellow.
      state : Int;
      "timer" : TON_TIME;
      timer_in : Bool;
      timer_q : Bool;
      first_scan : Bool := TRUE;
      wait_time : UInt;
   END_VAR
   VAR_TEMP
      "word" : Word;
      c : Int;
      error : Bool;
      tIdle : Bool;
      pt : Time;
   END_VAR
BEGIN
   // Aqualabo - Ponsel mesure
   // Dissolved oxygen (OPTOD), Conductivity (C4E, CTZ), pH_Redox, Turbi    
   // 
   // - Warning: For the oxygen sensor each pull for sensor measurement,
   //   will use of the available life span. Please set the measurement
   //   interval to appropriate value.
   // - Continuous assign true to start_measurement, to continuous do
   //   meassurements. #minimum_measurement_interval wil still restrict
   //   the interval time.
   // - https://en.aqualabo.fr/userfiles/doc/User%20Manual%20Oxygen%20Optical%20digital%20sensor%20OPTOD.pdf

   "mb_station_block_header"(sb := #sb,
                             mb_query := #mb_query);
   #mb_query.mb_addr := #mb_addr;
   #mb_query.mode := #mb_query.c.read.holding_reg;

   #"timer"(IN := #timer_in,
          PT := #"timer".PT,
          Q => #timer_q);
   #timer_in := false;

   IF #sb.out.Communication_error THEN // If communication error
       #state := 0;
       #Measurement_ok := false;
       #timer_in := true;  // Continue run the timer.
   ELSE
       CASE #state OF
           1:  // Compensate: Salinity, barometric pressure, temperature, etc.
               IF #compensate_enable THEN
                   #mb_query(mode := #mb_query.c.write.holding_reg,
                             data_addr := 16#5f,
                             data_ptr := #compensate);
                   #state += BOOL_TO_INT(#mb_query.Done);
               ELSE
                   #state += 1;
               END_IF;
           2:  // Read wait-time (Used later in state 4)
               #mb_query(data_addr := 16#A4,
                         data_ptr := #wait_time);
               #state += BOOL_TO_INT(#mb_query.Done);
           3:  // Start all meassurements.
               #"word" := 16#0f;
               #mb_query(mode := #mb_query.c.write.holding_reg,
                         data_addr := 16#01,
                         data_ptr := #"word");
               #state += BOOL_TO_INT(#mb_query.Done);
           4:  // Timer (Wait while sensor is obtaining measurements)
               #timer_in := true;
               PRESET_TIMER(TIMER := #"timer",
                            PT := MAX(IN1 := T_CONV(#wait_time),
                                      IN2 := T#1s)); // No less then 1s.
               #state += BOOL_TO_INT(#timer_q);
           5:  // Get data.
               #mb_query(data_addr := 16#0053,
                         data_ptr := #data1);
               // All measurements ok ?
               FOR #c := 0 TO 4 DO
                   #error := #error
                   OR #data1.status[#c].x00_Stm0
                   OR #data1.status[#c].x01_Stm1
                   OR #data1.status[#c].x02_Stm2;
               END_FOR;
               #Measurement_ok := NOT #error;
               IF #mb_query.Done THEN
                   // #start_measurement need to be assigned
                   // true again to start a new messurement.
                   #start_measurement := false;
                   #state := 0;
                   #QueryCnt += 1;
               END_IF;
           ELSE
               #tIdle := true;
               #timer_in := true;
               #pt := SEL(G := #api.interval = T#0s,
                          IN0 := #api.interval,
                          IN1 := #minimum_measurement_interval);
               PRESET_TIMER(PT := #pt,
                            TIMER := #"timer");

               #state := BOOL_TO_INT
               (NOT #api.wait AND // #api.wait may be set by other
                // function blocks to  halt the messurements.
                #start_measurement AND (
                (* *)#timer_q // Interval controlled
                (* *)OR #first_scan)); // At statup a messurement
               // is done as fast as possible.
       END_CASE;
   END_IF;
   // #wait is a API, for other blocks to stop the messurements,
   // #idle tells other blocks that no messurement is in progress.


   IF #sb.out.Communication_error
       OR #api.idle AND NOT #api.wait
   THEN
       // Description, Serial number, sw and hw version.
       #mb_query(data_addr := 3327,
                 data_ptr := #data2);
   END_IF;

   "mb_station_block_footer"(sb := #sb,
                             mb_query := #mb_query);

   #api.idle := #tIdle;
   #api.wait := false;
   #api.interval := T#0s;
   #first_scan := false;

   (* 
   Units:
   ---------------
   value0: Temperature
                         value1:                    value2:                    value3:       
   OPTOD (oxygen)    :   Oxygen [%Sat]              Oxygen [mg/l]              Oxygen [ppm]
   Turbi             :   Nephelo turbidity [NTU]    Nephelo turbidity [FNU]    TU turbidity [mg/L]
   pH_Redox          :   pH                         Redox [mV]
   conductivity_C4E  :   Conductivity C4E [uS/cm]   Salinity [ppt]             TDS - Kcl [ppm]
   Conductivity_CTZ  :   Conductivity CTZ [mS/cm]   Salinity [g/Kg]            Conductivity CTZ [mS/cm] 
                                                                               without temperature compensation                                                                  
   OPTOD: (Dissolved oxygen)
   Compensates[1]: Atmospheric pressure [hPa], default 1013 hPa
   Compensates[2]: Salinity [ppt], default 0 ppt


   Wiring: 
   Red     Wiring diagram V+
   black   Wiring diagram V-
   Green   B+ RS-485  (Siemens A)
   White   A- RS-485  (Siemens B)
   Blue    SDI-12

   Default settings:
   Buad: 9600
   Parity: none
   Modbus address: 10


   StmX:
   000: Measurement OK
   001: Measurement OK, but out of specifications
   010: Measurement OK with INFO 1 (See datasheet)
   011: Measurement OK with INFO 2 (See datasheet)
   100: Measurement impossible, out of specifications
   101: Measurement impossible with INFO 3 (See datasheet)
   110: Measurement impossible with INFO 4 (See datasheet)
   111: measurement under way (not yet available)

   StmGamme:       
   001: measurement used range 1
   010: measurement used range 2
   011: measurement used range 3
   100: measurement used range 4

   *)
END_FUNCTION_BLOCK

// folder: Library/Modbus/Station blocks/sb Tested/Schneider

FUNCTION_BLOCK "Schneider_enerlin_x_ife_lv43001"   // FB3, SCL
{ S7_Optimized_Access := 'TRUE' }
VERSION : 0.1
   VAR_INPUT
      mb_addr : USInt := 255;
   END_VAR
   VAR_IN_OUT
      mb_query : "mb_query";
   END_VAR
   VAR
      sb : "mb_station_block_udt";
      data : "energy_udt";
      "e" : Int;
      Frequency : Real;
   END_VAR
   VAR_TEMP
      param : "mb_set_udt";
      c : Int;
   END_VAR
   VAR CONSTANT
      ALL : DInt := 0;
   END_VAR
BEGIN
   // Schneider enerlin x ife iv43001 - Power meter gateway.
   // 
   // - Important : For tcp mb_addr need to be set to 255.
   //             : Timeout need to be set to at least 500ms, even on a local network.  
   // - 16#FFC0_0000 : Out of Order and Not Applicable Values
   //
   // DOCA0091EN-06
   // https://download.schneider-electric.com/files?p_Doc_Ref=DOCA0091EN
   //
   // There is a error in the datasheet, the addresses need to be subtracted by two.

   "mb_station_block_header"(sb := #sb, mb_query := #mb_query);
   #mb_query.mb_addr := #mb_addr;

   #mb_query.mode := #mb_query.c.read.holding_reg;

   IF "mb_query_range"(start := 32054, end := 32094, q := #mb_query) THEN
       #"e" += "mb_swap_word"(start := #ALL, end := #ALL, q := #mb_query);
       #"e" += "mb_read_buffer"(addr := 32056 - 2, ptr := #data.voltage.L_L, q := #mb_query);
       #"e" += "mb_read_buffer"(addr := 32068 - 2, ptr := #Frequency, q := #mb_query);
       #"e" += "mb_read_buffer"(addr := 32078 - 2, ptr := #data.power.active.total, q := #mb_query);
       #"e" += "mb_read_buffer"(addr := 32086 - 2, ptr := #data.power.reactive.total, q := #mb_query);
       #"e" += "mb_read_buffer"(addr := 32094 - 2, ptr := #data.power.apparent.total, q := #mb_query);

       // Invalid values: 16#FFC0_0000
       #"e" += "mb_read_buffer"(addr := 32062 - 2, ptr := #data.voltage.L_N, q := #mb_query);
       #"e" += "mb_read_buffer"(addr := 32072 - 2, ptr := #data.power.active.L, q := #mb_query);
       #"e" += "mb_read_buffer"(addr := 32080 - 2, ptr := #data.power.reactive.L, q := #mb_query);
   END_IF;

   (* // No values recived, maybe for other circuit breaker.
   IF "mb_query_range"(start := 12054 - 2, end := 12054 + 6, q := #mb_query) THEN
       #e += "mb_swap_word"(start := #ALL, end := #ALL, q := #mb_query);
       #e += "mb_read_buffer"(addr := 12054 - 2, ptr := #data.energy.active_received, q := #mb_query);
   END_IF; *)

   IF "mb_query_range"(start := 12015, end := 12017, q := #mb_query) THEN
       FOR #c := 1 TO 3 DO
           #data.current.L[#c] := "mb_buffer_get"(addr := 12015 + #c - 1, param := #param, q := #mb_query);
       END_FOR;
   END_IF;

   "mb_station_block_footer"(sb := #sb, mb_query := #mb_query);
END_FUNCTION_BLOCK

FUNCTION_BLOCK "Schneider_TRV00210"   // FB117, SCL
{ S7_Optimized_Access := 'TRUE' }
VERSION : 0.1
   VAR_INPUT
      mb_addr : USInt;
   END_VAR
   VAR_IN_OUT
      mb_query : "mb_query";
   END_VAR
   VAR
      sb : "mb_station_block_udt";
      data : "energy_udt";
      frequency : Real;
      power_factor : Struct
         L : Array[1..3] of Real;
         toal : Real;
      END_STRUCT;
   END_VAR
   VAR_TEMP
      c : Int;
      param : "mb_set_udt";
   END_VAR
BEGIN
   // Schneider - TRV00210 - Converter for power switches.
   //
   // 48940-328-01   06/2011
   //
   // - Not all register have values, and they are filled with 32768.
   // - If cable from circuit breaker is not connected, then every query will result in a exception.

   "mb_station_block_header"(sb := #sb, mb_query := #mb_query);
   #mb_query.mb_addr := #mb_addr;
   #mb_query.mode := #mb_query.c.read.holding_reg;
   #param.factor := 1;

   IF "mb_query_range"(start := 1046, end := 1053, q := #mb_query) THEN
       FOR #c := 1 TO 3 DO
           #power_factor.L[#c] := "mb_buffer_get"(addr := 1046 + #c - 1, param := #param, q := #mb_query);
       END_FOR;
       #power_factor.toal :="mb_buffer_get"(addr := 1049, param := #param, q := #mb_query);
       #frequency := "mb_buffer_get"(addr := 1053, param := #param, q := #mb_query) * 0.1;
   END_IF;

   IF "mb_query_range"(start := 12015, end := 12048, q := #mb_query) THEN
       FOR #c := 1 TO 3 DO
           #data.current.L[#c] := "mb_buffer_get"(addr := 12015 + #c - 1, param := #param, q := #mb_query);
           #data.voltage.L_L[#c] := "mb_buffer_get"(addr := 12029 + #c - 1, param := #param, q := #mb_query);
           #data.voltage.L_N[#c] := "mb_buffer_get"(addr := 12032 + #c - 1, param := #param, q := #mb_query);
           #data.power.active.L[#c] := "mb_buffer_get"(addr := 12037 + #c - 1, param := #param, q := #mb_query);
           #data.power.reactive.L[#c] := "mb_buffer_get"(addr := 12041 + #c - 1, param := #param, q := #mb_query);
           #data.power.apparent.L[#c] := "mb_buffer_get"(addr := 12045 + #c - 1, param := #param, q := #mb_query);
       END_FOR;
       #data.current.N := "mb_buffer_get"(addr := 12018, param := #param, q := #mb_query);
       #data.power.active.total := "mb_buffer_get"(addr := 12040, param := #param, q := #mb_query);
       #data.power.reactive.total := "mb_buffer_get"(addr := 12044, param := #param, q := #mb_query);
       #data.power.apparent.total := "mb_buffer_get"(addr := 12048, param := #param, q := #mb_query);
   END_IF;

   IF "mb_query_range"(start := 12053, end := 12066, q := #mb_query) THEN
       #param.double := true;
       #data.energy.active_in := "mb_buffer_get" (addr := 12053, param := #param, q := #mb_query);
       #data.energy.active_out := "mb_buffer_get"(addr := 12055, param := #param, q := #mb_query);
       #data.energy.reactive_in := "mb_buffer_get"(addr := 12057, param := #param, q := #mb_query);
       #data.energy.reactive_out := "mb_buffer_get"(addr := 12059, param := #param, q := #mb_query);
       #data.energy.apparent_in := "mb_buffer_get"(addr := 12063, param := #param, q := #mb_query);
       #data.energy.apparent_out := "mb_buffer_get"(addr := 12065, param := #param, q := #mb_query);
   END_IF;

   "mb_station_block_footer"(sb := #sb, mb_query := #mb_query);
END_FUNCTION_BLOCK

// folder: Library/Modbus/Station blocks/sb Tested/Siemens

FUNCTION_BLOCK "siemens_PAC3200"   // FB8, SCL
{ S7_Optimized_Access := 'TRUE' }
VERSION : 0.1
   VAR_INPUT
      mb_addr : USInt := 1;
   END_VAR
   VAR_IN_OUT
      mb_query : "mb_query";
   END_VAR
   VAR
      sb : "mb_station_block_udt";
      read1 : Struct
         voltage_L_n : Array[1..3] of Real;
         "voltage _L_L" : Array[1..3] of Real;   // 1:Va-b, 2:Vb-c, 3:Vc-a,
         current : Array[1..3] of Real;
         apparent_power : Array[1..3] of Real;
         active_power : Array[1..3] of Real;
         reactive_power : Array[1..3] of Real;
         power_factor : Array[1..3] of Real;
         THD_R_voltage : Array[1..3] of Real;
      END_STRUCT;
      read2 : Struct
         frequency : Real;   // unit: hz
         avg_voltage_Vph_n : Real;   // unit: V
         avg_voltage_Vph_ph : Real;   // unit: V
         avg_current : Real;   // unit: A
         total_apparent_power : Real;   // unit: VA
         total_active_power : Real;   // unit: W
      END_STRUCT;
   END_VAR
BEGIN
   // Siemens - PAC3200 - Power meter
   // 
   // Manual: 3.9.3, page 40

   "mb_station_block_header"(sb := #sb, mb_query := #mb_query);
   #mb_query.mb_addr := #mb_addr; // Device address.

   // Two queries, reading one section of holding registers each.
   #mb_query.mode := #mb_query.c.read.holding_reg;
   #mb_query(data_addr := 1, data_ptr := #read1);
   #mb_query(data_addr := 55, data_ptr := #read2);
   // - Each query reading one section of holding registers.
   // - Data length is automatically calculated for holding and input regisers.

   "mb_station_block_footer"(sb := #sb, mb_query := #mb_query);
END_FUNCTION_BLOCK

// folder: Library/Modbus/Station blocks/sb Untested

FUNCTION "readme_untested" : Void   // FC20, SCL
{ S7_Optimized_Access := 'TRUE' }
VERSION : 0.1
BEGIN
   (* The blocks in this folder is made with
      help of the datashett, no testing has 
      been done with equipment. Please 
      report bugs. 
   *)
END_FUNCTION

// folder: Library/Modbus/Station blocks/sb Untested/A

FUNCTION_BLOCK "Allen_bradley_power_flex_4"   // FB16, SCL
{ S7_Optimized_Access := 'TRUE' }
VERSION : 0.1
   VAR_INPUT
      mb_addr : USInt;
      ref : Real;
      reverse : Bool;
      reset : Bool;
   END_VAR
   VAR_OUTPUT
      Output_Frequency : Real;
      Output_Current : Real;
      DC_Bus_Voltage : Real;
      Output_Voltage : Real;
   END_VAR
   VAR_IN_OUT
      mb_query : "mb_query";
   END_VAR
   VAR
      sb : "mb_station_block_udt";
      read : Struct
         stat : Struct
            x08_At_Reference : Bool;
            x09_Reference_Controlled_by_Comm : Bool;
            x10_Operation_Cmd_Controlled_by_Comm : Bool;
            x11_Parameters_have_been_locked : Bool;
            x12_Digital_Input_1_Status : Bool;
            x13_Digital_Input_2_Status : Bool;
            x14 : Bool;
            x15 : Bool;
            "x00_Ready," : Bool;
            x01_Running : Bool;
            x02_cmd_Forward : Bool;
            x03_Rotating_Forward : Bool;
            x04_Accelerating : Bool;
            "x05_Decelerating," : Bool;
            x06_Alarm : Bool;
            x07_Faulted : Bool;
         END_STRUCT;
         error_code : UInt;
         ref_feedback : UInt;
         Output_Frequency : UInt;
         Output_Current : UInt;
         DC_Bus_Voltage : UInt;
         Output_Voltage : UInt;
      END_STRUCT;
      write : Struct
         cmd : Struct
            "x08_Accel Rate 1" : Bool := TRUE;
            "x09_Accel Rate 2" : Bool;
            "x10_Decel Rate 1" : Bool := TRUE;
            "x11_Decel Rate 2" : Bool;
            x12_Freq_Source_b0 : Bool := TRUE;
            x13_Freq_Source_b1 : Bool := TRUE;
            x14_Freq_Source_b2 : Bool;
            x15 : Bool;
            x00_Stop : Bool;
            x01_Start : Bool;
            x02_Jog : Bool;
            x03_Clear_Faults : Bool;
            x04_Forward : Bool;
            x05_Reverse : Bool;
            x06 : Bool;
            x07 : Bool;
         END_STRUCT;
         ref : UInt;
      END_STRUCT;
   END_VAR
BEGIN
   // Allen Bradley - Power Flex 4 - Compact AC Drive
   //
   // http://ab.rockwellautomation.com/Drives/PowerFlex-4
   // Web: https://plc-hmi-scadas.com/gallery/PowerFlex4ModBusAddressing.pdf

   "mb_station_block_header"(sb := #sb, mb_query := #mb_query);
   #mb_query.mb_addr := #mb_addr;

   #write.ref := REAL_TO_UINT(#ref * 10);
   #write.cmd.x00_Stop := #ref = 0;
   #write.cmd.x01_Start := #ref <> 0;
   #write.cmd.x03_Clear_Faults := #reset;
   #write.cmd.x04_Forward := NOT #reverse;
   #write.cmd.x05_Reverse := #reverse;

   #mb_query.mode := #mb_query.c.write.single_holding_reg;
   #mb_query(data_addr := 8192, data_ptr := #write.cmd);
   #mb_query(data_addr := 8193, data_ptr := #write.ref);

   #mb_query.mode := #mb_query.c.read.holding_reg;
   #mb_query(data_addr := 8448, data_ptr := #read);
   #Output_Frequency := UINT_TO_REAL(#read.Output_Frequency) / 10;
   #Output_Current := UINT_TO_REAL(#read.Output_Current) / 100;
   #DC_Bus_Voltage := UINT_TO_REAL(#read.DC_Bus_Voltage) / 10;
   #Output_Voltage := UINT_TO_REAL(#read.Output_Voltage) / 10;

   "mb_station_block_footer"(sb := #sb, mb_query := #mb_query);

   (* Error codes: (read.error_codes)
   0 - No Fault
   2 - Auxilary Input
   3 - Power Loss
   4 - Undervoltage
   5 - Overvoltage
   6 - Motor Stalled
   7 - Motor Overload
   8 - Heatsink Overtemperature
   12 - HW Overcurrent (300%)
   13 - Ground Fault
   29 - Analog Input Loss
   33 - Auto Restart Tries
   38 - Phase U to Ground Short
   39 - Phase V to Ground Short
   40 - Phase W to Ground Short
   41 - Phase U/V Short
   42 - Phase U/W Short
   43 - Phase V/W Short
   63 - Software Overcurrent
   64 - Drive Overload
   70 - Power Unit Fail
   80 - AutoTune Fail
   81 - Communication Loss
   100 - Parameter Checksum Error
   122 - I/O Board Fail         
   *)
END_FUNCTION_BLOCK

FUNCTION_BLOCK "Auma_valve"   // FB17, SCL
{ S7_Optimized_Access := 'TRUE' }
VERSION : 0.1
   VAR_INPUT
      mb_addr : UInt;
   END_VAR
   VAR_IN_OUT
      mb_query : "mb_query";
   END_VAR
   VAR
      sb : "mb_station_block_udt";
      read : Struct
         status : Struct
            torque_sw_closed : Bool;
            torque_sw_open : Bool;
            limit_sw_closed : Bool;
            limit_sw_open : Bool;
            sel_sw_local : Bool;
            sel_sw_remote : Bool;
            phase_fault : Bool;
            therminal_fault : Bool;
            falt : Bool;
            warning : Bool;
            running_close : Bool;
            running_open : Bool;
            not_ready_remote : Bool;
            setpoint_reached : Bool;
            end_p_clossed : Bool;
            end_p_open : Bool;
         END_STRUCT;
         "Actual position" : UInt;
      END_STRUCT;
      write : Struct
         cmd : Struct
            byte_2 : Byte;
            open : Bool;
            close : Bool;
            use_setpoint : Bool;
            reset : Bool;
            b4 : Bool;
            b5 : Bool;
            b6 : Bool;
            b7 : Bool;
         END_STRUCT;
         setpoint : UInt;
      END_STRUCT;
   END_VAR
BEGIN
   // Auma actuator controls
   // AC 01.2/ACExC 01.2 Modbus RTU
   //
   // http://www1.auma.com/uploads/media/sp_import2/handbuecher/
   // steuerungen/hb_ac2_modbus_geraeteintegration_en.pdf

   "mb_station_block_header"(sb := #sb, mb_query := #mb_query);
   #mb_query.mb_addr := #mb_addr;

   #mb_query(mode := #mb_query.c.read.input_reg,
             data_addr := 16#03E8,
             data_ptr := #read); // p.10

   #mb_query(mode := #mb_query.c.write.holding_reg,
             data_addr := 16#03E8,
             data_ptr := #write); // p.29

   "mb_station_block_footer"(sb := #sb, mb_query := #mb_query);

   (*
   - Each query reading one section of holding registers.
   - Data length is automatically calculated for holding 
     and input regisers.
   *)
END_FUNCTION_BLOCK

FUNCTION_BLOCK "Automatic_systems_AS1320"   // FB18, SCL
{ S7_Optimized_Access := 'TRUE' }
VERSION : 0.1
   VAR_INPUT
      mb_addr : UInt;
   END_VAR
   VAR_IN_OUT
      mb_query : "mb_query";
   END_VAR
   VAR
      sb : "mb_station_block_udt";
      read1 : Struct
         input : Word;
         input_3 : Word;
         output : Word;
         analog_in : Word;
         analog_out : Word;
         z2 : Array[1..4] of Word;
         temperature : Int;
         counter_1 : UDInt;
         counter_2 : UDInt;
         z : Array[1..3] of Word;
         state : Struct
            x08_blocked_closed : Bool;
            x09 : Bool;
            x10 : Bool;
            x11 : Bool;
            x12 : Bool;
            x13 : Bool;
            x14 : Bool;
            x15 : Bool;
            x00 : Bool;
            x01 : Bool;
            x02_open : Bool;
            x03_opening : Bool;
            x04_closed : Bool;
            x05_closing : Bool;
            x06_stop : Bool;
            x07_blocked_open : Bool;
         END_STRUCT;
      END_STRUCT;
      read2 : Struct
         PRDSTD : String[6];
         BL_xxx : String[6];
         "Type" : UInt;
         Change : UInt;
      END_STRUCT;
      write1 : Struct
         x08 : Bool;
         x09 : Bool;
         x10 : Bool;
         x11 : Bool;
         x12 : Bool;
         x13 : Bool;
         x14 : Bool;
         x15 : Bool;
         x00_open : Bool;
         x01_close : Bool;
         x02_block_open : Bool;
         x03_block_close : Bool;
         x04_stop : Bool;
         x05_reader_command_direction_a : Bool;
         x06_reader_command_direction_b : Bool;
         x07_reset_block : Bool;
      END_STRUCT;
      start_setup : Bool;
      write2 : Struct
         PS1_function : UInt;
         PS2_function : UInt;
         Positioning : UInt;
         barrier_type : UInt;
         arm_length : UInt;
         arm_type : UInt;
         power_fail_OP : UInt;
         exploitation : UInt;
      END_STRUCT;
      crank : Bool;
   END_VAR
BEGIN
   // Automatic systems - AS1320
   // http://www.visionbr.com.br/arquivo-produtos/20110823_92924_as1320-mt-en-16.pdf
   // Revision no: AS1320-prog 6.x-MT-FR-16 - 2009-11-10 

   "mb_station_block_header"(sb := #sb, mb_query := #mb_query);
   #mb_query.mb_addr := #mb_addr;

   #mb_query.mode := #mb_query.c.read.holding_reg;
   #mb_query(data_addr := 16#39, data_ptr := #read1);
   // #mb_query(data_addr := 16#00, data_ptr := #read3);
   // A micro switch at opening for the crank.
   #crank := #read1.input.%X14; 

   #mb_query.mode := #mb_query.c.write.holding_reg;
   #mb_query(data_addr := 16#12C, data_ptr := #write1);
   IF #start_setup THEN
       #mb_query(data_addr := 16#64, data_ptr := #write2);
       #start_setup := NOT #mb_query.Done;
   END_IF;

   "mb_station_block_footer"(sb := #sb, mb_query := #mb_query);
END_FUNCTION_BLOCK

FUNCTION_BLOCK "Accuenergy_Accuvim_L_Series_Power_meter"   // FB81, SCL
{ S7_Optimized_Access := 'TRUE' }
VERSION : 0.1
   VAR_INPUT
      mb_addr : USInt;
   END_VAR
   VAR_IN_OUT
      mb_query : "mb_query";
   END_VAR
   VAR
      sb : "mb_station_block_udt";
      read1 : Struct
         Frequency : Real;
         "Phase voltage" : Array[1..3] of Real;
         "Line voltage" : Array[1..3] of Real;
         Phase_current : Array[1..3] of Real;
         Neutral_current : Real;
         "Phase power" : Array[1..3] of Real;
         "System power Psum" : Real;
         "Phase reactive power" : Array[1..3] of Real;
         "System reactive power" : Real;
         "System apparent Ssum" : Real;
         Phase_power_factor : Array[1..3] of Real;
         "System power PFsum" : Real;
         "Voltage unbalance factor" : Real;
         "Current unbalance factor" : Real;
         _ : DWord;
         "Phase apparent power S" : Array[1..3] of Real;
         __ : DWord;
         "Apparent power demand" : Real;
         "Power demand P_Dmd" : Real;
         "Reactive power demand" : Real;
         "Phase current demand" : Array[1..3] of Real;
      END_STRUCT;
      read2_run_time : Struct
         Meter : UDInt;
         Load : UDInt;
      END_STRUCT;
      read3 : Struct
         Import_energy_Ep_imp : UDInt;
         Export_energy_Ep_exp : UDInt;
         Import_reactive_energy_Eq_imp : UDInt;
         Export_reactive_energy_Eq_exp : UDInt;
         Apparent_energy_Es : UDInt;
         Phase_energy : Array[1..3] of Struct
            "import Ep_imp" : UDInt;
            "export Ep_exp" : UDInt;
         END_STRUCT;
      END_STRUCT;
   END_VAR
BEGIN
   // Accuenergy - Accuvim-L Series Power meter
   // 
   // - https://www.accuenergy.com/files/acuvim-l/
   //   Acuvim-L-Panel-Submeter-Power-Energy-Meter-User-%20Manual(1030E2201).pdf

   "mb_station_block_header"(sb := #sb, mb_query := #mb_query);
   #mb_query.mb_addr := #mb_addr;

   #mb_query.mode := #mb_query.c.read.holding_reg;
   #mb_query(data_addr := 16#600, data_ptr := #read1);
   #mb_query(data_addr := 16#180, data_ptr := #read2_run_time);
   #mb_query(data_addr := 16#156, data_ptr := #read3);

   "mb_station_block_footer"(sb := #sb, mb_query := #mb_query);
END_FUNCTION_BLOCK

// folder: Library/Modbus/Station blocks/sb Untested/A/Abb

FUNCTION_BLOCK "abb_aquaMaster_3"   // FB4, SCL
{ S7_Optimized_Access := 'TRUE' }
VERSION : 0.1
   VAR_INPUT
      mb_addr : USInt;
   END_VAR
   VAR_IN_OUT
      mb_query : "mb_query";
   END_VAR
   VAR
      sb : "mb_station_block_udt";
      flow : Real;
      pressure : Real;
      totaliser : Struct
         fwd : DInt;
         rev : DInt;
         net : DInt;
      END_STRUCT;
   END_VAR
BEGIN
   // - ABB - AquaMaster 3 - Electromagnetic flowmeter
   // - COI/FET2XX/MOD/TBLÃ¢â‚¬â€œEN
   // - https://library.e.abb.com/public/
   //   91eead459bb0d349c12577fc0033d2b5/COI_FET2XX_MOD_TBL-EN.pdf

   "mb_station_block_header"(sb := #sb, mb_query := #mb_query);
   #mb_query.mb_addr := #mb_addr; // Device address.

   // Two queries, reading input registers. 
   #mb_query.mode := #mb_query.c.read.input_reg;
   #mb_query(data_addr := 5017, data_ptr := #flow);
   #mb_query(data_addr := 5025, data_ptr := #pressure);

   // One query, reading one section of holding registers.
   #mb_query.mode := #mb_query.c.read.holding_reg;
   #mb_query(data_addr := 12003, data_ptr := #totaliser);

   // - Each query reading one section of holding registers.
   // - Data length is automatically calculated for holding 
   //   and input regisers.

   "mb_station_block_footer"(sb := #sb, mb_query := #mb_query);
END_FUNCTION_BLOCK

FUNCTION_BLOCK "Abb_266"   // FB12, SCL
{ S7_Optimized_Access := 'TRUE' }
VERSION : 0.1
   VAR_INPUT
      mb_addr : UInt;
   END_VAR
   VAR_IN_OUT
      mb_query : "mb_query";
   END_VAR
   VAR
      sb : "mb_station_block_udt";
      data : Struct
         "Differential Pressure" : Real;
         "Static Pressure" : Real;
         "Process Temperature" : Real;
         "Mass flow rate value" : Real;
         "Volume Flow rate value" : Real;
      END_STRUCT;
      settings : Struct
         Differential_Pressure_Units_Code : UInt := 12;
         Static_Pressure_Units_select_Code : UInt := 12;
         Temperature_Units_select_Code : UInt := 32;
      END_STRUCT;
   END_VAR
BEGIN
   // ABB - 266 MODBUS, multivariable transmitter.
   // Differential and Static Pressure, Temperature
   // 
   // https://library.e.abb.com/public/9b5a1233ec79400387d5b4887002fb00/2105216MNAA.pdf

   "mb_station_block_header"(sb := #sb, mb_query := #mb_query);
   #mb_query.mb_addr := #mb_addr;

   #mb_query(mode := #mb_query.c.read.holding_reg,
             data_addr := 401,
             data_ptr := #data);

   #mb_query(mode := #mb_query.c.write.holding_reg,
             data_addr := 481,
             data_ptr := #settings);

   "mb_station_block_footer"(sb := #sb, mb_query := #mb_query);

   (*
   Differential_Pressure_Units_Code
   1 = inches of water
   8 = Millibar (ROM default)
   11 = Pascal
   12 = Kilopascal 

   Static Pressure Units select Code
   6 = PSIA
   7 = Bar (ROM default)
   12 = Kilopascal
   117 = Megapascal 

   Temperature Units select Code
   32 = Degree Celsius (ROM default)
   33 = Degree Fahrenheit
   34 = Degree Rankine
   35 = Degree Kelvin

   *)
END_FUNCTION_BLOCK

FUNCTION_BLOCK "Abb_M2M_DMTME"   // FB15, SCL
{ S7_Optimized_Access := 'TRUE' }
VERSION : 0.1
   VAR_INPUT
      mb_addr : UInt;
   END_VAR
   VAR_IN_OUT
      mb_query : "mb_query";
   END_VAR
   VAR
      sb : "mb_station_block_udt";
      read1 : Struct
         "3-PHASE SYSTEM VOLTAGE" : UDInt;   // volt
         voltage_Lx_N : Array[1..3] of UDInt;   // volt
         voltage_L_L : Array[1..3] of UDInt;   // volt 1:L1-L2, 2:L2-L3, 3:L3-L1
         "3-PHASE SYSTEM CURRENT" : UDInt;
         current : Array[1..3] of UDInt;   // mA
         "3-PHASE SYS. POWER FACTOR" : DInt;   // x1000
         Power_factor : Array[1..3] of DInt;   // x1000
         "3-PHASE SYSTEM COS Ï•I" : DInt;   // x1000
         phase_cos : Array[1..3] of DInt;   // x1000
      END_STRUCT;
      read2 : Struct
         "3-PHASE S. APPARENT POWER" : UDInt;   // VA
         apparent_power : Array[1..3] of UDInt;   // VA
         "3-PHASE SYS. ACTIVE POWER" : DInt;   // Watt
         active_power : Array[1..3] of DInt;   // Watt
         "3-PHASE S. REACTIVE POWER" : UDInt;
         reactive_power : Array[1..3] of UDInt;
         "3-PHASE SYS. ACTIVE ENERGY" : UDInt;   // Wh * 100
         "3-PHASE S. REACTIVE ENERGY" : UDInt;   // VArh * 100
         frequency : UDInt;   // mHz
         "MAX LINE CURRENT" : Array[1..3] of UDInt;
      END_STRUCT;
   END_VAR
BEGIN
   // ABB - M2M/DMTME - 2CSG445011D0201 
   //
   // https://library.e.abb.com/public/3921770555944801ad6d9e002d23ca23/2CSG445011D0201.pdf

   "mb_station_block_header"(sb := #sb, mb_query := #mb_query);
   #mb_query.mb_addr := #mb_addr;

   #mb_query.mode := #mb_query.c.read.holding_reg;
   #mb_query(data_addr := 16#1000, data_ptr := #read1);
   #mb_query(data_addr := 16#1026, data_ptr := #read2);

   "mb_station_block_footer"(sb := #sb, mb_query := #mb_query);
END_FUNCTION_BLOCK

FUNCTION_BLOCK "Abb_ach_400_ac_drives"   // FB80, SCL
{ S7_Optimized_Access := 'TRUE' }
VERSION : 0.1
   VAR_INPUT
      mb_addr : UInt;
   END_VAR
   VAR_IN_OUT
      mb_query : "mb_query";
   END_VAR
   VAR
      sb : "mb_station_block_udt";
      read1 : Struct
         sw : Struct   // page 111, tabel 23
            x08_actual_eq_ref : Bool;   // (= is within tolerance limits)
            x09_drive_control_remote : Bool;
            x10_supervision_limit : Bool;   // The value of first supervised parameter equals to or is greater than supervision limit. Refer toGroup 32 Supervision.
            x11_ext2_selected : Bool;   // 0 = ext1 selected
            x12_run : Bool;   // Enable signal received
            x13 : Bool;
            x14 : Bool;
            x15 : Bool;
            x00_rdy_to_sw_on : Bool;
            x01_rdy_to_operate : Bool;
            x02_opr_enabled : Bool;
            x03_falut : Bool;
            x04_OFF2_inactive : Bool;
            x05_OFF3_inactive : Bool;
            x06_switch_on_innhibited : Bool;
            x07_alarm : Bool;   // See the Diagnostics section for a list of relevant alarms
         END_STRUCT;
      END_STRUCT;
      read2 : Struct
         speed : Int;   // rpm
         output_freq : Int;   // 0.1 Hz
         current : Int;   // 0.1 A
         torque : Int;   // 0.1 %
         power : Int;   // 0.1 kW
         dc_bus_voltage : Int;   // 0.1 V
         output_voltage : Int;   // 0.1 V
         ACH400_temp : Int;   // 0.1 Â°C | Displays the temperature of the ACH 400 heatsink in degrees Centigrade
         ext_ref_1 : Int;   // 0.1 Hz
         ext_ref_2 : Int;   // 0.1 %
         ctrl_location : Int;   // 0 - 2
         run_time : UInt;   // h
         kWh_cnt : UInt;   // kWh
         appl_blk_output : UInt;
         digital_input : Struct
            x08 : Bool;
            x09 : Bool;
            x10 : Bool;
            x11 : Bool;
            x12 : Bool;
            x13 : Bool;
            x14 : Bool;
            x15 : Bool;
            x00_in_1 : Bool;
            x01_in_2 : Bool;
            x02_in_3 : Bool;
            x03_in_4 : Bool;
            x04 : Bool;
            x05 : Bool;
            x06 : Bool;
            x07 : Bool;
         END_STRUCT;
         analog_in_1 : UInt;   // 0.1 %
         analog_in_2 : UInt;   // 0.1 %
      END_STRUCT;
      read3 : Struct
         fault_word_1 : Struct
            x08_Motor_overtemperature : Bool;
            x09_Panel_loss : Bool;
            x10_Parameters_inconsistent : Bool;
            x11_DC_bus_ripple_too_large : Bool;
            x12_Motor_stall : Bool;
            x13_Serial_communication_loss : Bool;
            x14_External_fault : Bool;
            x15_Output_ground_fault : Bool;
            x00_Overcurrent : Bool;
            x01_DC_overvoltage : Bool;
            x02_ACH_400_overtemperature : Bool;
            x03_Fault_current : Bool;
            x04_Output_overload : Bool;
            x05_DC_undervoltage : Bool;
            x06_Analog_input_1_fault : Bool;
            x07_Analog_input_2_fault : Bool;
         END_STRUCT;
         fault_word_2 : Struct
            x08_hw_err : Bool;
            x09_hw_err : Bool;
            x10_hw_err : Bool;
            x11_hw_err : Bool;
            x12_hw_err : Bool;
            x13_hw_err : Bool;
            x14_hw_err : Bool;
            x15_hw_err : Bool;
            x00_Underload : Bool;
            x01 : Bool;
            x02_DDCS_link : Bool;
            x03 : Bool;
            x04 : Bool;
            x05 : Bool;
            x06 : Bool;
            x07 : Bool;
         END_STRUCT;
      END_STRUCT;
      _ : Bool;
      write1 : Struct
         cw : Struct   // page 109, tabel 21
            x08 : Bool;
            x09 : Bool;
            x10 : Bool;
            x11_sel_ext_2 : Bool;   // Select external control location 1
            x12 : Bool;
            x13 : Bool;
            x14 : Bool;
            x15 : Bool;
            x00_start : Bool := TRUE;
            x01_no_cost_stop : Bool := TRUE;   // Emergency OFF, coast to stop.Enter OFF2 ACTIVE; proceed to SWITCH-ON INHIBITED
            x02_no_ramp_stop : Bool := TRUE;   // Emergency stop. Drive ramps to stop according to parameter 2205 DECELER TIME 2. Enter
            x03_operation_enable : Bool := TRUE;
            x04 : Bool;
            x05_no_ramp_generator : Bool := TRUE;
            x06_no_force_ramp_generator_input2zero : Bool;   // Force Ramp Function Generator input to zero
            x07_fault_reset : Bool;   // (enter SWITCH-ON INHIBITED)
         END_STRUCT;
         ref_1 : Int;
         ref_2 : Int;
      END_STRUCT;
      write2 : Struct
         keypad_ref_sel : UInt;
         ext1_ext2_sel : UInt;
         ext1_sel : UInt;
         ext1_sel_min : UInt;   // 0 - 250 Hz
         ext1_sel_max : UInt := 50;   // 0 - 250 Hz
      END_STRUCT;
      write3 : Struct   // Communication fault function
         comm_fault_func : UInt := 1;   // 1=FAULT(cost), 2=CONST SP 7, 3=LAST SPEED
      END_STRUCT;
   END_VAR
BEGIN
   // Abb - ACH 400 - AC Drives 
   // 
   // Web: https://www.ccontrols.com/support/dp/ACH402_US_04_Web.pdf

   "mb_station_block_header"(sb := #sb, mb_query := #mb_query);
   #mb_query.mb_addr := #mb_addr;

   #mb_query.mode := #mb_query.c.read.holding_reg;
   #mb_query(data_addr := 3, data_ptr := #read1);   // 40004
   #mb_query(data_addr := 102, data_ptr := #read2); // 103
   #mb_query(data_addr := 304, data_ptr := #read3); // 305 - 1 

   #mb_query.mode := #mb_query.c.write.holding_reg;
   #mb_query(data_addr := 0, data_ptr := #write1); // 40001
   // #mb_query(data_addr := 1100, data_ptr := #write2); // 1101 - 1
   #mb_query(data_addr := 5003, data_ptr := #write3); // 5004 - 1

   "mb_station_block_footer"(sb := #sb, mb_query := #mb_query);
END_FUNCTION_BLOCK

// folder: Library/Modbus/Station blocks/sb Untested/B

FUNCTION_BLOCK "Belimo_vav_Compact_mod"   // FB19, SCL
{ S7_Optimized_Access := 'TRUE' }
VERSION : 0.1
   VAR_INPUT
      mb_addr : UInt;
      sp : Real;   // setpoint
      bus_fail_position : Real;
   END_VAR
   VAR_OUTPUT
      pos_feedback : Real;
   END_VAR
   VAR_IN_OUT
      mb_query : "mb_query";
   END_VAR
   VAR
      sb : "mb_station_block_udt";
      read : Struct
         position : Int;
      END_STRUCT;
      write1 : Struct
         setpoint : Int;
      END_STRUCT;
      write2 : Struct
         bus_fail_position : Int;
      END_STRUCT;
   END_VAR
BEGIN
   // Belimo - VAV-Compact MOD 
   // LMV-D3-MOD 5  Nm 2   W 4 VA (max. 5 A @ 5 ms) Approx. 500 g
   // NMV-D3-MOD 10 Nm 3.5 W 6 VA (max. 5 A @ 5 ms) Approx. 700 g
   // https://www.micromatic.no/globalassets/inriver/
   // resources/ko1070_0_5_1.pdf

   "mb_station_block_header"(sb := #sb, mb_query := #mb_query);
   #mb_query.mb_addr := #mb_addr;

   #mb_query.mode := #mb_query.c.read.holding_reg;
   #mb_query(data_addr := 4, data_ptr := #read);
   #pos_feedback := INT_TO_REAL(#read.position) * 0.01;

   #mb_query.mode := #mb_query.c.write.holding_reg;
   #write1.setpoint := REAL_TO_INT(#sp) * 100;
   #mb_query(data_addr := 0, data_ptr := #write1);
   #write2.bus_fail_position := REAL_TO_INT(#bus_fail_position) * 100;
   #mb_query(data_addr := 108, data_ptr := #write2);

   "mb_station_block_footer"(sb := #sb, mb_query := #mb_query);

   (*
   Bus fail position:
   0 Last setpoint (no bus monitoring)
   1 Fast close if time is exceeded
   2 Fast open if time is exceeded 
   *)
END_FUNCTION_BLOCK

FUNCTION_BLOCK "Binmaster_mnu_ultrasonic_sensor"   // FB20, SCL
{ S7_Optimized_Access := 'TRUE' }
VERSION : 0.1
   VAR_INPUT
      mb_addr : UInt;
   END_VAR
   VAR_IN_OUT
      mb_query : "mb_query";
   END_VAR
   VAR
      sb : "mb_station_block_udt";
      data : Struct
         "Model Type" : UInt;
         Raw_Distance_Level : UInt;   // [mm]
         _ : UInt;
         Temperature : Int;
         Calculated : DInt;
         __ : DWord;
         "Version" : UInt;
         "Signal Strength" : UInt;
         ___ : UInt;
         "Trip 1 Alarm" : UInt;
         "Trip 1 Status" : UInt;
         "Trip 2 Alarm" : UInt;
         "Trip 2 Status" : UInt;
      END_STRUCT;
      setting : Struct
         Units : UInt := 3;   // 3=Meters
         Distance : Struct
            Max : UInt;   // 0 - 15,250 mm
            Full : UInt;   // 0 - 15,250 mm
            Empty : UInt;
         END_STRUCT;
         cal : Struct
            Multiplier : UInt := 1000;   // 1000 -> 1.000
            Offset : UInt := 0;
         END_STRUCT;
      END_STRUCT;
   END_VAR
BEGIN
   // Binmaster - MNU Ultrasonic Sensor
   // 
   // Web: http://www.binmaster.com/_resources/e30d:ogspbx-on/files/
   // 75651567z4d4b98f5/_fn/BinMaster%20MNU%20manual%209004257%20Rev%20A1.pdf

   "mb_station_block_header"(sb := #sb, mb_query := #mb_query);
   #mb_query.mb_addr := #mb_addr;

   #mb_query.mode := #mb_query.c.mode.read;
   #mb_query(data_addr := 30299, data_ptr := #data);

   #mb_query.mode := #mb_query.c.mode.write;
   #mb_query(data_addr := 40401, data_ptr := #setting.Units);
   #mb_query(data_addr := 40405, data_ptr := #setting.Distance);
   #mb_query(data_addr := 40416, data_ptr := #setting.cal);

   "mb_station_block_footer"(sb := #sb, mb_query := #mb_query);
END_FUNCTION_BLOCK

// folder: Library/Modbus/Station blocks/sb Untested/D

FUNCTION_BLOCK "Delta_CFP2000"   // FB22, SCL
{ S7_Optimized_Access := 'TRUE' }
VERSION : 0.1
   VAR_INPUT
      mb_addr : USInt;
      ref : Real;   // (minus=>rev.)
   END_VAR
   VAR_OUTPUT
      stat : Struct
         drive_stops : Bool;
         drive_decelerating : Bool;
         drive_standby : Bool;
         drive_operating : Bool;
      END_STRUCT;
      current : Real;
   END_VAR
   VAR_IN_OUT
      mb_query : "mb_query";
   END_VAR
   VAR
      sb : "mb_station_block_udt";
      read : Struct
         warn_code : USInt;
         error_code : USInt;
         stat : Struct
            "b08_Master frequency controlled by communication" : Bool;
            "b09 Master frequency controlled by analog signal" : Bool;
            "b10 Operation command controlled by communication interface" : Bool;
            "b11 Parameter locked" : Bool;
            "b12 Enable to copy parameters from keypad" : Bool;
            b13 : Bool;
            b14 : Bool;
            b15 : Bool;
            b00_oper_stat : Bool;
            b01_oper_stat : Bool;
            b02 : Bool;
            b03_direction : Bool;
            b04_direction : Bool;
            b05 : Bool;
            b06 : Bool;
            b07 : Bool;
         END_STRUCT;
         frequency_cmd : Int;
         output_frequency : Int;
         output_current : UInt;
         "DC-BUS Voltage" : UInt;
         output_voltage : UInt;
         "Current step number of Multi-Step Speed Operation" : Int;
         _ : Int;
         counter_value : Int;
         power_factor_angle : Int;
         output_torque : Int;
         actual_motor_speed : Int;
         __ : Int;
         ___ : Int;
         power_output : Int;   // kwh
      END_STRUCT;
      write : Struct
         cmd_word : Struct
            b08_sel_speed : Bool;
            b09_sel_speed : Bool;
            b10_sel_speed : Bool;
            b11_sel_speed : Bool;
            b12_Enable_bit06_11_function : Bool := TRUE;
            b13_oper_keypad : Bool;
            b14_oper_Pr_00_21_setting : Bool;
            b15 : Bool;
            b00_stop : Bool;
            b01_run : Bool;
            b02 : Bool;
            b03 : Bool;
            b04_fwd : Bool;
            b05_rev : Bool;
            b06_sel_accel_decel : Bool;
            b07_sel_accel_decel : Bool;
         END_STRUCT;
         ref_freq : UInt;
         "a" : Struct
            b08 : Bool;
            b09 : Bool;
            b10 : Bool;
            b11 : Bool;
            b12 : Bool;
            b13 : Bool;
            b14 : Bool;
            b15 : Bool;
            b00_external_fault : Bool;
            b01_reset : Bool;
            b02_B_B_ON : Bool;
            b03 : Bool;
            b04 : Bool;
            b05 : Bool;
            b06 : Bool;
            b07 : Bool;
         END_STRUCT;
      END_STRUCT;
   END_VAR
BEGIN
   // Delta - CFP2000 - Variable frequency drive
   // 
   // http://www.softstartuk.com/wp-content/uploads/2017/07/VFD-CFP2000_UM_EN_20170303.pdf

   "mb_station_block_header"(sb := #sb, mb_query := #mb_query);
   #mb_query.mb_addr := #mb_addr;

   // Read
   #mb_query.mode := #mb_query.c.read.holding_reg;

   #mb_query(data_addr := 16#2100, data_ptr := #read);
   #stat.drive_stops := NOT #read.stat.b00_oper_stat AND NOT #read.stat.b01_oper_stat;
   #stat.drive_decelerating := #read.stat.b00_oper_stat AND NOT #read.stat.b01_oper_stat;
   #stat.drive_standby := NOT #read.stat.b00_oper_stat AND #read.stat.b01_oper_stat;
   #stat.drive_operating := #read.stat.b00_oper_stat AND #read.stat.b01_oper_stat;
   #current := UINT_TO_REAL(#read.output_current) * 100;
   // Output current (XX.XX A). When current is higher than
   // 655.35, it will shift decimal as (XXX.XA). The decimal
   // can refer to High byte of 211F. 

   // Write
   #mb_query.mode := #mb_query.c.write.holding_reg;

   #write.ref_freq := REAL_TO_UINT(#ref * 100);
   #write.cmd_word.b00_stop := #ref = 0;
   #write.cmd_word.b01_run := NOT #write.cmd_word.b00_stop;
   #write.cmd_word.b05_rev := #ref < 0;
   #write.cmd_word.b04_fwd := NOT #write.cmd_word.b05_rev;
   #mb_query(data_addr := 16#2000, data_ptr := #write);

   "mb_station_block_footer"(sb := #sb, mb_query := #mb_query);
END_FUNCTION_BLOCK

FUNCTION_BLOCK "DAE_Instrument_PM210"   // FB82, SCL
{ S7_Optimized_Access := 'TRUE' }
VERSION : 0.1
   VAR_INPUT
      mb_addr : USInt;
   END_VAR
   VAR_IN_OUT
      mb_query : "mb_query";
   END_VAR
   VAR
      sb : "mb_station_block_udt";
   END_VAR
   VAR RETAIN
      conf : Struct
         write : Bool;
         PT_ratio : Real;
         CT_ratio : Real;
      END_STRUCT;
   END_VAR
   VAR
      data1 : Struct
         voltage_Lx_N : Array[1..3] of Real;
         voltage_L_L : Array[1..3] of Real;
         current : Array[1..3] of Real;
         total_active_power : Real;
         total_reactive_power : Real;
         total_apparent_power : Real;
         frequency : Real;
         power_factor : Real;
         total_active_energy : Real;
         total_reactive_energy : Real;
         "15_minute_block_demand" : Real;
         "1_minute_block_demand" : Real;
         generator_total_active_energy : Real;
         generator_total_reactive_energy : Real;
      END_STRUCT;
      data2 : Struct
         energy_active : Struct   // VA
            phase : Array[1..3] of Real;
            total : Real;
         END_STRUCT;
         energy_reactive : Struct
            phase : Array[1..3] of Real;
            total : Real;
         END_STRUCT;
         power_active : Struct
            phase : Array[1..3] of Real;
            total : Real;
         END_STRUCT;
         power_reactive : Struct
            phase : Array[1..3] of Real;
            total : Real;
         END_STRUCT;
         power_apparent : Struct
            phase : Array[1..3] of Real;
            total : Real;
         END_STRUCT;
         power_factor : Struct
            phase : Array[1..3] of Real;
            total : Real;
         END_STRUCT;
      END_STRUCT;
      read3_temperature : Int;
      read4_io : Struct
         digital_output : Word;
         digital_input : Word;
      END_STRUCT;
      data5_generator_energy : Struct
         active : Struct
            phase : Array[1..3] of Real;
            total : Real;
         END_STRUCT;
         reactive : Struct
            phase : Array[1..3] of Real;
            total : Real;
         END_STRUCT;
      END_STRUCT;
   END_VAR
   VAR_TEMP
      read1 : Struct
         voltage_Lx_N : Array[1..3] of UDInt;   // volt
         voltage_L_L : Array[1..3] of UDInt;   // volt 1:L1-L2, 2:L2-L3, 3:L3-L1
         current : Array[1..3] of UDInt;   // mA
         total_active_power : UDInt;
         total_reactive_power : UDInt;
         total_apparent_power : UDInt;
         frequency : UDInt;
         power_factor : DInt;
         total_active_energy : UDInt;
         total_reactive_energy : UDInt;
         "15_minute_block_demand" : UDInt;
         "1_minute_block_demand" : UDInt;
         generator_total_active_energy : UDInt;
         generator_total_reactive_energy : UDInt;
      END_STRUCT;
      read2 : Struct
         energy_active : Struct   // VA
            phase : Array[1..3] of UDInt;
            total : UDInt;
         END_STRUCT;
         energy_reactive : Struct
            phase : Array[1..3] of UDInt;
            total : UDInt;
         END_STRUCT;
         power_active : Struct
            phase : Array[1..3] of UDInt;
            total : UDInt;
         END_STRUCT;
         power_reactive : Struct
            phase : Array[1..3] of UDInt;
            total : UDInt;
         END_STRUCT;
         power_apparent : Struct
            phase : Array[1..3] of UDInt;
            total : UDInt;
         END_STRUCT;
         power_factor : Struct
            phase : Array[1..3] of Int;
            total : Int;
         END_STRUCT;
      END_STRUCT;
      read5_generator_energy : Struct
         active : Struct
            phase : Array[1..3] of UDInt;
            total : UDInt;
         END_STRUCT;
         reactive : Struct
            phase : Array[1..3] of UDInt;
            total : UDInt;
         END_STRUCT;
      END_STRUCT;
      write1 : Struct
         PT_ratio : UInt;
         CT_ratio : UInt;
      END_STRUCT;
      c : Int;
   END_VAR
BEGIN
   // DAE Instrument Corp. - PM210 
   // Multi-Function Panel Meter
   //
   // Default: 9600-8-N-1
   // 
   // http://www.daeinstrument.com/downloads/PM210%20Modbus%20Reference-2.6.1e.pdf

   "mb_station_block_header"(sb := #sb, mb_query := #mb_query);
   #mb_query.mb_addr := #mb_addr;
   #mb_query.mode := #mb_query.c.read.holding_reg;

   #mb_query(data_addr := 20, data_ptr := #read1);
   IF #mb_query.Done THEN
       FOR #c := 1 TO 3 DO
           #data1.voltage_Lx_N[#c] := UDINT_TO_REAL(ROR(IN := #read1.voltage_Lx_N[#c], N := 16)) * 0.1;
           #data1.voltage_L_L[#c] := UDINT_TO_REAL(ROR(IN := #read1.voltage_L_L[#c], N := 16)) * 0.1;
           #data1.current[#c] := UDINT_TO_REAL(ROR(IN := #read1.current[#c], N := 16)) * 0.001;
       END_FOR;
       #data1.total_active_power := UDINT_TO_REAL(ROR(IN := #read1.total_active_power, N := 16));
       #data1.total_reactive_power := UDINT_TO_REAL(ROR(IN := #read1.total_reactive_power, N := 16));
       #data1.total_apparent_power := UDINT_TO_REAL(ROR(IN := #read1.total_apparent_power, N := 16));
       #data1.frequency := UDINT_TO_REAL(ROR(IN := #read1.frequency, N := 16)) * 0.1;
       #data1.power_factor := DINT_TO_REAL(ROR(IN := #read1.power_factor, N := 16)) * 0.001;
       #data1.total_active_energy := UDINT_TO_REAL(ROR(IN := #read1.total_active_energy, N := 16)) * 0.01;
       #data1.total_reactive_energy := UDINT_TO_REAL(ROR(IN := #read1.total_reactive_energy, N := 16)) * 0.01;
       #data1."15_minute_block_demand" := UDINT_TO_REAL(ROR(IN := #read1."15_minute_block_demand", N := 16)) * 0.1;
       #data1."1_minute_block_demand" := UDINT_TO_REAL(ROR(IN := #read1."1_minute_block_demand", N := 16)) * 0.1;
       #data1.generator_total_active_energy := UDINT_TO_REAL(ROR(IN := #read1.generator_total_active_energy, N := 16)) * 0.01;
       #data1.generator_total_reactive_energy := UDINT_TO_REAL(#read1.generator_total_reactive_energy) * 0.01;
   END_IF;

   #mb_query(data_addr := 80, data_ptr := #read2);
   IF #mb_query.Done THEN
       FOR #c := 1 TO 3 DO
           #data2.energy_active.phase[#c] := UDINT_TO_REAL(ROR(IN := #read2.energy_active.phase[#c], N := 16)) * 0.01;
           #data2.energy_reactive.phase[#c] := UDINT_TO_REAL(ROR(IN := #read2.energy_reactive.phase[#c], N := 16)) * 0.01;
           #data2.power_active.phase[#c] := UDINT_TO_REAL(ROR(IN := #read2.power_active.phase[#c], N := 16));
           #data2.power_reactive.phase[#c] := UDINT_TO_REAL(ROR(IN := #read2.power_reactive.phase[#c], N := 16));
           #data2.power_apparent.phase[#c] := UDINT_TO_REAL(ROR(IN := #read2.power_apparent.phase[#c], N := 16));
           #data2.power_factor.phase[#c] := INT_TO_REAL(#read2.power_factor.phase[#c]) * 0.001;
       END_FOR;
       #data2.energy_active.total := UDINT_TO_REAL(ROR(IN := #read2.energy_active.total, N := 16)) * 0.01;
       #data2.energy_reactive.total := UDINT_TO_REAL(ROR(IN := #read2.energy_reactive.total, N := 16)) * 0.01;
       #data2.power_active.total := UDINT_TO_REAL(ROR(IN := #read2.power_active.total, N := 16));
       #data2.power_reactive.total := UDINT_TO_REAL(ROR(IN := #read2.power_reactive.total, N := 16));
       #data2.power_apparent.total := UDINT_TO_REAL(ROR(IN := #read2.power_apparent.total, N := 16));
       #data2.power_factor.total := INT_TO_REAL(#read2.power_factor.total) * 0.001;
   END_IF;

   #mb_query(data_addr := 139, data_ptr := #read3_temperature);
   #mb_query(data_addr := 142, data_ptr := #read4_io);
   #mb_query(data_addr := 144, data_ptr := #read5_generator_energy);
   IF #mb_query.Done THEN
       FOR #c := 1 TO 3 DO
           #data5_generator_energy.active.phase[#c] := UDINT_TO_REAL(ROR(IN := #read5_generator_energy.active.phase[#c], N := 16)) * 0.01;
           #data5_generator_energy.reactive.phase[#c] := UDINT_TO_REAL(ROR(IN := #read5_generator_energy.reactive.phase[#c], N := 16)) * 0.01;
       END_FOR;
       #data5_generator_energy.active.total := UDINT_TO_REAL(ROR(IN := #read5_generator_energy.active.total, N := 16)) * 0.01;
       #data5_generator_energy.reactive.total := UDINT_TO_REAL(ROR(IN := #read5_generator_energy.reactive.total, N := 16)) * 0.01;
   END_IF;

   IF #conf.write THEN
       #write1.PT_ratio := REAL_TO_UINT(#conf.PT_ratio * 100);
       #write1.CT_ratio := REAL_TO_UINT(#conf.CT_ratio);
       #mb_query(mode := #mb_query.c.write.holding_reg,
                 data_addr := 133,
                 data_ptr := #write1);
       #conf.write := #conf.write AND NOT #mb_query.Done;
   END_IF;

   "mb_station_block_footer"(sb := #sb, mb_query := #mb_query);
END_FUNCTION_BLOCK

// folder: Library/Modbus/Station blocks/sb Untested/E

FUNCTION_BLOCK "Emerson_Micro_Motion"   // FB23, SCL
{ S7_Optimized_Access := 'TRUE' }
VERSION : 0.1
   VAR_INPUT
      mb_addr : UInt;
   END_VAR
   VAR_IN_OUT
      mb_query : "mb_query";
   END_VAR
   VAR
      sb : "mb_station_block_udt";
      data : Struct
         stat : Struct
            x08_Primary_mA_output_saturated : Bool;
            x09_Secondary_mA_output_saturated : Bool;
            x10_Primary_mA_output_fixed : Bool;
            x11_Secondary_mA_output_fixed : Bool;
            x12_Density_overrange : Bool;
            x13_Flowmeter_zeroing_failure : Bool;
            x14_Zero_value_too_low : Bool;
            x15_Zero_value_too_high : Bool;
            x00_EPROM_checksum_failure : Bool;
            x01_RAM_diagnostic_failure : Bool;
            x02_Sensor_failure : Bool;
            x03_Temperature_sensor_failure : Bool;
            x04_Input_overrange : Bool;
            x05_Frequency_pulse_output_saturated : Bool;
            x06_Transmitter_not_configured : Bool;
            x07_Realtime_interrupt_failure : Bool;
            x24 : Bool;
            x25 : Bool;
            x26 : Bool;
            x27 : Bool;
            x28 : Bool;
            x29 : Bool;
            x30 : Bool;
            x31 : Bool;
            x16_Transmitter_electronics_failure : Bool;
            x17_Flowmeter_zeroing_in_progress : Bool;
            x18_Slug_flow : Bool;
            x19_Power_reset_occurred : Bool;
            x20_Transmitter_configuration_changed : Bool;
            x21_Transmitter_initializing_warming_up : Bool;
            x22 : Bool;
            x23 : Bool;
         END_STRUCT;
         "Mass flow rate" : Real;
         Density : Real;
         Temperature : Real;
         "Volume flow rate" : Real;
         Pressure : Real;   // (internally derived)
         "Mass total" : Real;
         "Volume total" : Real;
         "Mass inventory" : Real;
         "Volume inventory" : Real;
      END_STRUCT;
   END_VAR
BEGIN
   // Emerson - Micro Motion Transmitters
   // RFT9739, MVD DC, Modeo 1500, Model 1700, Model 2500, Model 2700, Series 3000
   // 
   // http://www2.emersonprocess.com/siteadmincenter/PM%20Micro%20Motion%20Documents/Modbus-Map-Manual-20001741.pdf

   "mb_station_block_header"(sb := #sb, mb_query := #mb_query);
   #mb_query.mb_addr := #mb_addr;

   #mb_query.mode := #mb_query.c.read.holding_reg;
   #mb_query(data_addr := 245, data_ptr := #data);

   "mb_station_block_footer"(sb := #sb, mb_query := #mb_query);
END_FUNCTION_BLOCK

FUNCTION_BLOCK "Endress_proline_promass_83"   // FB24, SCL
{ S7_Optimized_Access := 'TRUE' }
VERSION : 0.1
   VAR_INPUT
      mb_addr : UInt;
   END_VAR
   VAR_OUTPUT
      device_ok : Bool;
   END_VAR
   VAR_IN_OUT
      mb_query : "mb_query";
   END_VAR
   VAR
      sb : "mb_station_block_udt";
      data : Struct
         mass_flow : Real;
         temperature : Real;
         totalizer : Real;
         actual_system_condition : Int;   // 1->ok
      END_STRUCT;
   END_VAR
BEGIN
   // Endress - Proline Promass 83
   // Web: https://portal.endress.com/wa001/dla/5000000/5862/000/05/BA00107DEN_1311.pdf

   "mb_station_block_header"(sb := #sb, mb_query := #mb_query);
   #mb_query.mb_addr := #mb_addr;

   #mb_query(mode := #mb_query.c.read.holding_reg,
             data_addr := 5051,
             data_ptr := #data);

   "mb_station_block_footer"(sb := #sb, mb_query := #mb_query);

   #device_ok := #data.actual_system_condition = 1;
END_FUNCTION_BLOCK

FUNCTION_BLOCK "Epluse_EE071"   // FB25, SCL
{ S7_Optimized_Access := 'TRUE' }
VERSION : 0.1
   VAR_INPUT
      mb_addr : USInt := 247;
   END_VAR
   VAR_IN_OUT
      mb_query : "mb_query";
   END_VAR
   VAR
      sb : "mb_station_block_udt";
      data : Struct
         temperature_C : Real;   // [Â°C]
         temperature_F : Real;   // [Â°F]
         humidity_rel : Real;   // [%]
         humidity_abs : Real;   // [g/mÂ³]
      END_STRUCT;
      serial : String[8];
   END_VAR
BEGIN
   // Epluse - EE071
   // Humidity and Temperature Probe
   //
   // http://downloads.epluse.com/fileadmin/data/product/ee071/datasheet_EE071.pdf

   "mb_station_block_header"(sb := #sb, mb_query := #mb_query);
   #mb_query.mb_addr := #mb_addr;

   #mb_query.mode := #mb_query.c.read.holding_reg;
   #mb_query(data_addr := 30026, data_ptr := #data);
   #mb_query(data_addr := 30001, data_ptr := #serial); // 30001-30008

   "mb_station_block_footer"(sb := #sb, mb_query := #mb_query);

   (*IF #sb.out.communication_error THEN
       #data.temperature_C := 0;
       #data.temperature_F := 0;
       #data.humidity_rel := 0;
       #data.humidity_abs := 0;
   END_IF;*)

   (* Electrical connections

   Supply voltage 1) 2) 4 - 28 V DC

   brown...+UB
   white.....B-RS485 (= Data-)
   blue......A-RS485 (= Data+)
   black....GND
   grey......shielding

   1...+UB
   2...B-RS485 (= Data-)
   3...A-RS485 (= Data+)
   4...GND

   *)
END_FUNCTION_BLOCK

